LIN {X 0,Y 137.983,Z 516.99,A -85,B 0,C 180,E1 -24854.754,E2 -24854.754} C_VEL
LIN {X 0,Y 141.442,Z 522.73,A -85,B 0,C 180,E1 -24860.354,E2 -24860.354} C_VEL
LIN {X 0,Y 146.281,Z 527.08,A -85,B 0,C 180,E1 -24865.62,E2 -24865.62} C_VEL
LIN {X 0,Y 152.76,Z 530.196,A -85,B 0,C 180,E1 -24870.403,E2 -24870.403} C_VEL
LIN {X 0,Y 160.519,Z 532.095,A -85,B 0,C 180,E1 -24874.693,E2 -24874.693} C_VEL
LIN {X 0,Y 169.487,Z 532.782,A -85,B 0,C 180,E1 -24878.462,E2 -24878.462} C_VEL
LIN {X 0,Y 179.412,Z 532.227,A -85,B 0,C 180,E1 -24881.754,E2 -24881.754} C_VEL
LIN {X 0,Y 184.679,Z 531.482,A -85,B 0,C 180,E1 -24883.235,E2 -24883.235} C_VEL
LIN {X 0,Y 184.884,Z 531.53,A -85,B 0,C 180,E1 -24883.757,E2 -24883.757} C_VEL
LIN {X 0,Y 174.334,Z 533.909,A -85,B 0,C 180,E1 -24886.736,E2 -24886.736} C_VEL
LIN {X 0,Y 164.676,Z 535.155,A -85,B 0,C 180,E1 -24890.193,E2 -24890.193} C_VEL
LIN {X 0,Y 156.139,Z 535.296,A -85,B 0,C 180,E1 -24894.184,E2 -24894.184} C_VEL
LIN {X 0,Y 149.124,Z 534.399,A -85,B 0,C 180,E1 -24898.771,E2 -24898.771} C_VEL
LIN {X 0,Y 143.456,Z 532.415,A -85,B 0,C 180,E1 -24903.835,E2 -24903.835} C_VEL
LIN {X 0,Y 139.272,Z 529.177,A -85,B 0,C 180,E1 -24909.698,E2 -24909.698} C_VEL
LIN {X 0,Y 136.298,Z 533.394,A -85,B 0,C 180,E1 -24914.345,E2 -24914.345} C_VEL
LIN {X 0,Y 134.877,Z 535.787,A -85,B 0,C 180,E1 -24917.967,E2 -24917.967} C_VEL
LIN {X 0,Y 134.143,Z 537.216,A -85,B 0,C 180,E1 -24920.954,E2 -24920.954} C_VEL
LIN {X 0,Y 133.779,Z 538.232,A -85,B 0,C 180,E1 -24923.966,E2 -24923.966} C_VEL
LIN {X 0,Y 133.683,Z 538.88,A -85,B 0,C 180,E1 -24927.125,E2 -24927.125} C_VEL
LIN {X 0,Y 132.985,Z 539.095,A -85,B 0,C 180,E1 -24929.635,E2 -24929.635} C_VEL
LIN {X 0,Y 131.345,Z 538.952,A -85,B 0,C 180,E1 -24932.112,E2 -24932.112} C_VEL
LIN {X 0,Y 127.673,Z 537.738,A -85,B 0,C 180,E1 -24937.168,E2 -24937.168} C_VEL
LIN {X 0,Y 126.865,Z 536.758,A -85,B 0,C 180,E1 -24939.814,E2 -24939.814} C_VEL
LIN {X 0,Y 126.909,Z 536.327,A -85,B 0,C 180,E1 -24940.702,E2 -24940.702} C_VEL
LIN {X 0,Y 128.167,Z 533.463,A -85,B 0,C 180,E1 -24945.909,E2 -24945.909} C_VEL
LIN {X 0,Y 130.287,Z 529.76,A -85,B 0,C 180,E1 -24950.522,E2 -24950.522} C_VEL
LIN {X 0,Y 133.208,Z 524.928,A -85,B 0,C 180,E1 -24954.962,E2 -24954.962} C_VEL
LIN {X 0,Y 137.32,Z 517.944,A -85,B 0,C 180,E1 -24959.745,E2 -24959.745} C_VEL
LIN {X 0,Y 141.86,Z 509.751,A -85,B 0,C 180,E1 -24963.869,E2 -24963.869} C_VEL
LIN {X 0,Y 146.119,Z 501.674,A -85,B 0,C 180,E1 -24966.954,E2 -24966.954} C_VEL
LIN {X 0,Y 150.862,Z 491.823,A -85,B 0,C 180,E1 -24969.829,E2 -24969.829} C_VEL
LIN {X 0,Y 155.426,Z 480.689,A -85,B 0,C 180,E1 -24972.265,E2 -24972.265} C_VEL
LIN {X 0,Y 159.193,Z 469.804,A -85,B 0,C 180,E1 -24974.049,E2 -24974.049} C_VEL
LIN {X 0,Y 162.606,Z 457.774,A -85,B 0,C 180,E1 -24975.488,E2 -24975.488} C_VEL
LIN {X 0,Y 165.253,Z 444.892,A -85,B 0,C 180,E1 -24976.554,E2 -24976.554} C_VEL
LIN {X 0,Y 166.908,Z 431.8,A -85,B 0,C 180,E1 -24977.266,E2 -24977.266} C_VEL
LIN {X 0,Y 169.217,Z 398.153,A -85,B 0,C 180,E1 -24978.515,E2 -24978.515} C_VEL
LIN {X 0,Y 168.56,Z 385.284,A -85,B 0,C 180,E1 -24979.583,E2 -24979.583} C_VEL
LIN {X 0,Y 163.304,Z 375.445,A -85,B 0,C 180,E1 -24982.466,E2 -24982.466} C_VEL
LIN {X 0,Y 157.969,Z 366.553,A -85,B 0,C 180,E1 -24985.731,E2 -24985.731} C_VEL
LIN {X 0,Y 153.227,Z 359.41,A -85,B 0,C 180,E1 -24989.031,E2 -24989.031} C_VEL
LIN {X 0,Y 150.396,Z 355.476,A -85,B 0,C 180,E1 -24991.238,E2 -24991.238} C_VEL
LIN {X 0,Y 147.419,Z 351.407,A -85,B 0,C 180,E1 -24993.833,E2 -24993.833} C_VEL
LIN {X 0,Y 144.792,Z 348.208,A -85,B 0,C 180,E1 -24996.394,E2 -24996.394} C_VEL
LIN {X 0,Y 143.823,Z 346.644,A -85,B 0,C 180,E1 -24997.481,E2 -24997.481} C_VEL
LIN {X 0,Y 141.32,Z 344.263,A -85,B 0,C 180,E1 -25000.386,E2 -25000.386} C_VEL
LIN {X 0,Y 139.709,Z 341.234,A -85,B 0,C 180,E1 -25002.81,E2 -25002.81} C_VEL
LIN {X 0,Y 136.958,Z 339.298,A -85,B 0,C 180,E1 -25007.403,E2 -25007.403} C_VEL
LIN {X 0,Y 135.502,Z 336.05,A -85,B 0,C 180,E1 -25011.518,E2 -25011.518} C_VEL
LIN {X 0,Y 135.356,Z 335.408,A -85,B 0,C 180,E1 -25012.167,E2 -25012.167} C_VEL
LIN {X 0,Y 134.092,Z 334.839,A -85,B 0,C 180,E1 -25020,E2 -25020} C_VEL
LIN {X 0,Y 135.381,Z 335.546,A -85,B 0,C 180,E1 -25028.396,E2 -25028.396} C_VEL
LIN {X 0,Y 136.672,Z 338.936,A -85,B 0,C 180,E1 -25032.416,E2 -25032.416} C_VEL
LIN {X 0,Y 138.936,Z 340.918,A -85,B 0,C 180,E1 -25036.531,E2 -25036.531} C_VEL
LIN {X 0,Y 139.96,Z 341.514,A -85,B 0,C 180,E1 -25038.007,E2 -25038.007} C_VEL
LIN {X 0,Y 141.534,Z 344.542,A -85,B 0,C 180,E1 -25040.34,E2 -25040.34} C_VEL
LIN {X 0,Y 144.237,Z 347.153,A -85,B 0,C 180,E1 -25043.417,E2 -25043.417} C_VEL
LIN {X 0,Y 146.603,Z 350.647,A -85,B 0,C 180,E1 -25045.88,E2 -25045.88} C_VEL
LIN {X 0,Y 148.083,Z 352.258,A -85,B 0,C 180,E1 -25047.217,E2 -25047.217} C_VEL
LIN {X 0,Y 150.906,Z 356.018,A -85,B 0,C 180,E1 -25049.611,E2 -25049.611} C_VEL
LIN {X 0,Y 155.786,Z 363.227,A -85,B 0,C 180,E1 -25053.258,E2 -25053.258} C_VEL
LIN {X 0,Y 161.121,Z 371.713,A -85,B 0,C 180,E1 -25056.699,E2 -25056.699} C_VEL
LIN {X 0,Y 166.735,Z 381.737,A -85,B 0,C 180,E1 -25059.903,E2 -25059.903} C_VEL
LIN {X 0,Y 170.224,Z 388.868,A -85,B 0,C 180,E1 -25061.746,E2 -25061.746} C_VEL
LIN {X 0,Y 167.52,Z 425.77,A -85,B 0,C 180,E1 -25063.139,E2 -25063.139} C_VEL
LIN {X 0,Y 165.601,Z 439.061,A -85,B 0,C 180,E1 -25064.047,E2 -25064.047} C_VEL
LIN {X 0,Y 162.942,Z 451.365,A -85,B 0,C 180,E1 -25065.288,E2 -25065.288} C_VEL
LIN {X 0,Y 160.167,Z 461.584,A -85,B 0,C 180,E1 -25066.72,E2 -25066.72} C_VEL
LIN {X 0,Y 156.593,Z 471.955,A -85,B 0,C 180,E1 -25068.552,E2 -25068.552} C_VEL
LIN {X 0,Y 152.311,Z 482.567,A -85,B 0,C 180,E1 -25071.05,E2 -25071.05} C_VEL
LIN {X 0,Y 147.955,Z 492.24,A -85,B 0,C 180,E1 -25074.077,E2 -25074.077} C_VEL
LIN {X 0,Y 143.542,Z 500.604,A -85,B 0,C 180,E1 -25077.417,E2 -25077.417} C_VEL
LIN {X 0,Y 139.074,Z 508.063,A -85,B 0,C 180,E1 -25081.313,E2 -25081.313} C_VEL
LIN {X 0,Y 135.383,Z 514.04,A -85,B 0,C 180,E1 -25085.466,E2 -25085.466} C_VEL
LIN {X 0,Y 132.292,Z 518.76,A -85,B 0,C 180,E1 -25089.803,E2 -25089.803} C_VEL
LIN {X 0,Y 129.919,Z 522.361,A -85,B 0,C 180,E1 -25094.311,E2 -25094.311} C_VEL
LIN {X 0,Y 128.741,Z 524.212,A -85,B 0,C 180,E1 -25097.391,E2 -25097.391} C_VEL
LIN {X 0,Y 127.826,Z 525.621,A -85,B 0,C 180,E1 -25100.509,E2 -25100.509} C_VEL
LIN {X 0,Y 126.857,Z 527.214,A -85,B 0,C 180,E1 -25106.827,E2 -25106.827} C_VEL
LIN {X 0,Y 126.763,Z 527.441,A -85,B 0,C 180,E1 -25110.003,E2 -25110.003} C_VEL
LIN {X 0,Y 127.085,Z 526.871,A -85,B 0,C 180,E1 -25115.478,E2 -25115.478} C_VEL
LIN {X 0,Y 127.815,Z 525.69,A -85,B 0,C 180,E1 -25119.498,E2 -25119.498} C_VEL
LIN {X 0,Y 128.715,Z 524.32,A -85,B 0,C 180,E1 -25122.619,E2 -25122.619} C_VEL
LIN {X 0,Y 130.56,Z 521.447,A -85,B 0,C 180,E1 -25127.224,E2 -25127.224} C_VEL
LIN {X 0,Y 133.185,Z 517.529,A -85,B 0,C 180,E1 -25131.681,E2 -25131.681} C_VEL
LIN {X 0,Y 136.479,Z 512.452,A -85,B 0,C 180,E1 -25135.961,E2 -25135.961} C_VEL
LIN {X 0,Y 140.425,Z 506.047,A -85,B 0,C 180,E1 -25140.035,E2 -25140.035} C_VEL
LIN {X 0,Y 145.115,Z 498.061,A -85,B 0,C 180,E1 -25143.848,E2 -25143.848} C_VEL
LIN {X 0,Y 149.172,Z 489.824,A -85,B 0,C 180,E1 -25146.958,E2 -25146.958} C_VEL
LIN {X 0,Y 153.639,Z 479.82,A -85,B 0,C 180,E1 -25149.825,E2 -25149.825} C_VEL
LIN {X 0,Y 157.58,Z 469.857,A -85,B 0,C 180,E1 -25151.993,E2 -25151.993} C_VEL
LIN {X 0,Y 161.097,Z 458.996,A -85,B 0,C 180,E1 -25153.836,E2 -25153.836} C_VEL
LIN {X 0,Y 164.233,Z 446.902,A -85,B 0,C 180,E1 -25155.354,E2 -25155.354} C_VEL
LIN {X 0,Y 166.651,Z 433.829,A -85,B 0,C 180,E1 -25156.511,E2 -25156.511} C_VEL
LIN {X 0,Y 168.152,Z 421.523,A -85,B 0,C 180,E1 -25157.195,E2 -25157.195} C_VEL
LIN {X 0,Y 170.406,Z 389.046,A -85,B 0,C 180,E1 -25158.395,E2 -25158.395} C_VEL
LIN {X 0,Y 165.265,Z 378.802,A -85,B 0,C 180,E1 -25161.152,E2 -25161.152} C_VEL
LIN {X 0,Y 160.009,Z 369.693,A -85,B 0,C 180,E1 -25164.252,E2 -25164.252} C_VEL
LIN {X 0,Y 155.37,Z 362.549,A -85,B 0,C 180,E1 -25167.317,E2 -25167.317} C_VEL
LIN {X 0,Y 153.571,Z 359.786,A -85,B 0,C 180,E1 -25168.63,E2 -25168.63} C_VEL
LIN {X 0,Y 153.009,Z 359.751,A -85,B 0,C 180,E1 -25168.982,E2 -25168.982} C_VEL
LIN {X 0,Y 151.499,Z 361.411,A -85,B 0,C 180,E1 -25169.798,E2 -25169.798} C_VEL
LIN {X 0,Y 147.778,Z 373.075,A -85,B 0,C 180,E1 -25171.215,E2 -25171.215} C_VEL
LIN {X 0,Y 145.671,Z 378.207,A -85,B 0,C 180,E1 -25172.233,E2 -25172.233} C_VEL
LIN {X 0,Y 143.605,Z 381.544,A -85,B 0,C 180,E1 -25173.484,E2 -25173.484} C_VEL
LIN {X 0,Y 142.496,Z 382.609,A -85,B 0,C 180,E1 -25174.277,E2 -25174.277} C_VEL
LIN {X 0,Y 138.592,Z 397.916,A -85,B 0,C 180,E1 -25175.899,E2 -25175.899} C_VEL
LIN {X 0,Y 135.86,Z 407.043,A -85,B 0,C 180,E1 -25177.372,E2 -25177.372} C_VEL
LIN {X 0,Y 134.347,Z 410.966,A -85,B 0,C 180,E1 -25178.419,E2 -25178.419} C_VEL
LIN {X 0,Y 133.86,Z 411.757,A -85,B 0,C 180,E1 -25178.841,E2 -25178.841} C_VEL
LIN {X 0,Y 133.459,Z 411.859,A -85,B 0,C 180,E1 -25179.279,E2 -25179.279} C_VEL
LIN {X 0,Y 133.201,Z 410.793,A -85,B 0,C 180,E1 -25179.741,E2 -25179.741} C_VEL
LIN {X 0,Y 133.317,Z 407.838,A -85,B 0,C 180,E1 -25180.162,E2 -25180.162} C_VEL
LIN {X 0,Y 132.531,Z 426.85,A -85,B 0,C 180,E1 -25182.345,E2 -25182.345} C_VEL
LIN {X 0,Y 131.767,Z 440.893,A -85,B 0,C 180,E1 -25184.533,E2 -25184.533} C_VEL
LIN {X 0,Y 131.039,Z 452.449,A -85,B 0,C 180,E1 -25186.876,E2 -25186.876} C_VEL
LIN {X 0,Y 130.192,Z 465.708,A -85,B 0,C 180,E1 -25190.288,E2 -25190.288} C_VEL
LIN {X 0,Y 129.673,Z 476.575,A -85,B 0,C 180,E1 -25193.777,E2 -25193.777} C_VEL
LIN {X 0,Y 129.296,Z 486.462,A -85,B 0,C 180,E1 -25197.663,E2 -25197.663} C_VEL
LIN {X 0,Y 129.201,Z 494.658,A -85,B 0,C 180,E1 -25201.558,E2 -25201.558} C_VEL
LIN {X 0,Y 129.288,Z 502.752,A -85,B 0,C 180,E1 -25206.241,E2 -25206.241} C_VEL
LIN {X 0,Y 130.06,Z 510.449,A -85,B 0,C 180,E1 -25211.691,E2 -25211.691} C_VEL
LIN {X 0,Y 132.13,Z 516.795,A -85,B 0,C 180,E1 -25217.009,E2 -25217.009} C_VEL
LIN {X 0,Y 136.037,Z 522.64,A -85,B 0,C 180,E1 -25222.797,E2 -25222.797} C_VEL
LIN {X 0,Y 139.975,Z 526.09,A -85,B 0,C 180,E1 -25226.864,E2 -25226.864} C_VEL
LIN {X 0,Y 146.71,Z 529.673,A -85,B 0,C 180,E1 -25231.799,E2 -25231.799} C_VEL
LIN {X 0,Y 154.737,Z 532.05,A -85,B 0,C 180,E1 -25236.189,E2 -25236.189} C_VEL
LIN {X 0,Y 163.997,Z 533.24,A -85,B 0,C 180,E1 -25240.002,E2 -25240.002} C_VEL
LIN {X 0,Y 174.202,Z 533.221,A -85,B 0,C 180,E1 -25243.302,E2 -25243.302} C_VEL
LIN {X 0,Y 174.544,Z 533.221,A -85,B 0,C 180,E1 -25243.547,E2 -25243.547} C_VEL
LIN {X 0,Y 164.125,Z 534.493,A -85,B 0,C 180,E1 -25246.751,E2 -25246.751} C_VEL
LIN {X 0,Y 153.064,Z 534.613,A -85,B 0,C 180,E1 -25251.312,E2 -25251.312} C_VEL
LIN {X 0,Y 146.693,Z 533.865,A -85,B 0,C 180,E1 -25254.903,E2 -25254.903} C_VEL
LIN {X 0,Y 140.065,Z 532.02,A -85,B 0,C 180,E1 -25259.88,E2 -25259.88} C_VEL
LIN {X 0,Y 134.974,Z 529.091,A -85,B 0,C 180,E1 -25265.38,E2 -25265.38} C_VEL
LIN {X 0,Y 133.476,Z 527.79,A -85,B 0,C 180,E1 -25267.657,E2 -25267.657} C_VEL
LIN {X 0,Y 129.895,Z 532.5,A -85,B 0,C 180,E1 -25272.685,E2 -25272.685} C_VEL
LIN {X 0,Y 127.936,Z 535.47,A -85,B 0,C 180,E1 -25277.303,E2 -25277.303} C_VEL
LIN {X 0,Y 127.137,Z 536.899,A -85,B 0,C 180,E1 -25280.451,E2 -25280.451} C_VEL
LIN {X 0,Y 126.721,Z 537.916,A -85,B 0,C 180,E1 -25283.628,E2 -25283.628} C_VEL
LIN {X 0,Y 126.611,Z 538.647,A -85,B 0,C 180,E1 -25287.651,E2 -25287.651} C_VEL
LIN {X 0,Y 126.759,Z 538.767,A -85,B 0,C 180,E1 -25289.997,E2 -25289.997} C_VEL
LIN {X 0,Y 126.546,Z 538.522,A -85,B 0,C 180,E1 -25293.18,E2 -25293.18} C_VEL
LIN {X 0,Y 126.756,Z 536.845,A -85,B 0,C 180,E1 -25299.571,E2 -25299.571} C_VEL
LIN {X 0,Y 126.909,Z 536.327,A -85,B 0,C 180,E1 -25300.702,E2 -25300.702} C_VEL
LIN {X 0,Y 126.775,Z 535.087,A -85,B 0,C 180,E1 -25303.305,E2 -25303.305} C_VEL
LIN {X 0,Y 125.297,Z 532.462,A -85,B 0,C 180,E1 -25307.605,E2 -25307.605} C_VEL
LIN {X 0,Y 124.449,Z 529.896,A -85,B 0,C 180,E1 -25311.042,E2 -25311.042} C_VEL
LIN {X 0,Y 124.853,Z 527.661,A -85,B 0,C 180,E1 -25313.555,E2 -25313.555} C_VEL
LIN {X 0,Y 125.292,Z 526.84,A -85,B 0,C 180,E1 -25314.356,E2 -25314.356} C_VEL
LIN {X 0,Y 129.229,Z 520.714,A -85,B 0,C 180,E1 -25319.301,E2 -25319.301} C_VEL
LIN {X 0,Y 133.556,Z 513.613,A -85,B 0,C 180,E1 -25323.537,E2 -25323.537} C_VEL
LIN {X 0,Y 138.648,Z 504.783,A -85,B 0,C 180,E1 -25327.461,E2 -25327.461} C_VEL
LIN {X 0,Y 143.436,Z 495.72,A -85,B 0,C 180,E1 -25330.479,E2 -25330.479} C_VEL
LIN {X 0,Y 148.106,Z 485.642,A -85,B 0,C 180,E1 -25333.006,E2 -25333.006} C_VEL
LIN {X 0,Y 152.465,Z 474.478,A -85,B 0,C 180,E1 -25335.127,E2 -25335.127} C_VEL
LIN {X 0,Y 156.222,Z 462.931,A -85,B 0,C 180,E1 -25336.734,E2 -25336.734} C_VEL
LIN {X 0,Y 159.321,Z 450.322,A -85,B 0,C 180,E1 -25337.985,E2 -25337.985} C_VEL
LIN {X 0,Y 161.652,Z 436.707,A -85,B 0,C 180,E1 -25338.862,E2 -25338.862} C_VEL
LIN {X 0,Y 164.022,Z 407.003,A -85,B 0,C 180,E1 -25340.003,E2 -25340.003} C_VEL
LIN {X 0,Y 164.518,Z 398.539,A -85,B 0,C 180,E1 -25340.36,E2 -25340.36} C_VEL
LIN {X 0,Y 163.994,Z 388.51,A -85,B 0,C 180,E1 -25341.257,E2 -25341.257} C_VEL
LIN {X 0,Y 158.892,Z 378.792,A -85,B 0,C 180,E1 -25344.317,E2 -25344.317} C_VEL
LIN {X 0,Y 153.534,Z 369.735,A -85,B 0,C 180,E1 -25347.947,E2 -25347.947} C_VEL
LIN {X 0,Y 149.787,Z 364.14,A -85,B 0,C 180,E1 -25350.822,E2 -25350.822} C_VEL
LIN {X 0,Y 147.92,Z 361.462,A -85,B 0,C 180,E1 -25352.403,E2 -25352.403} C_VEL
LIN {X 0,Y 145.368,Z 357.807,A -85,B 0,C 180,E1 -25354.783,E2 -25354.783} C_VEL
LIN {X 0,Y 142.706,Z 354.313,A -85,B 0,C 180,E1 -25357.575,E2 -25357.575} C_VEL
LIN {X 0,Y 141.994,Z 353.199,A -85,B 0,C 180,E1 -25358.422,E2 -25358.422} C_VEL
LIN {X 0,Y 139.451,Z 350.415,A -85,B 0,C 180,E1 -25361.64,E2 -25361.64} C_VEL
LIN {X 0,Y 138.378,Z 348.166,A -85,B 0,C 180,E1 -25363.4,E2 -25363.4} C_VEL
LIN {X 0,Y 135.587,Z 345.861,A -85,B 0,C 180,E1 -25368.457,E2 -25368.457} C_VEL
LIN {X 0,Y 134.268,Z 342.408,A -85,B 0,C 180,E1 -25372.859,E2 -25372.859} C_VEL
LIN {X 0,Y 133.228,Z 341.881,A -85,B 0,C 180,E1 -25380,E2 -25380} C_VEL
LIN {X 0,Y 134.331,Z 342.692,A -85,B 0,C 180,E1 -25387.894,E2 -25387.894} C_VEL
LIN {X 0,Y 135.726,Z 346.121,A -85,B 0,C 180,E1 -25392.333,E2 -25392.333} C_VEL
LIN {X 0,Y 138.44,Z 348.337,A -85,B 0,C 180,E1 -25397.162,E2 -25397.162} C_VEL
LIN {X 0,Y 140.391,Z 351.729,A -85,B 0,C 180,E1 -25400.114,E2 -25400.114} C_VEL
LIN {X 0,Y 142.392,Z 353.705,A -85,B 0,C 180,E1 -25402.49,E2 -25402.49} C_VEL
LIN {X 0,Y 144.806,Z 357.248,A -85,B 0,C 180,E1 -25405.13,E2 -25405.13} C_VEL
LIN {X 0,Y 146.115,Z 358.845,A -85,B 0,C 180,E1 -25406.389,E2 -25406.389} C_VEL
LIN {X 0,Y 149.396,Z 363.613,A -85,B 0,C 180,E1 -25409.311,E2 -25409.311} C_VEL
LIN {X 0,Y 152.868,Z 368.804,A -85,B 0,C 180,E1 -25412.027,E2 -25412.027} C_VEL
LIN {X 0,Y 157.952,Z 377.189,A -85,B 0,C 180,E1 -25415.539,E2 -25415.539} C_VEL
LIN {X 0,Y 163.364,Z 387.261,A -85,B 0,C 180,E1 -25418.839,E2 -25418.839} C_VEL
LIN {X 0,Y 165.441,Z 391.583,A -85,B 0,C 180,E1 -25420.019,E2 -25420.019} C_VEL
LIN {X 0,Y 162.744,Z 426.104,A -85,B 0,C 180,E1 -25421.319,E2 -25421.319} C_VEL
LIN {X 0,Y 160.761,Z 439.35,A -85,B 0,C 180,E1 -25422.234,E2 -25422.234} C_VEL
LIN {X 0,Y 157.996,Z 451.663,A -85,B 0,C 180,E1 -25423.484,E2 -25423.484} C_VEL
LIN {X 0,Y 155.097,Z 461.888,A -85,B 0,C 180,E1 -25424.93,E2 -25424.93} C_VEL
LIN {X 0,Y 151.362,Z 472.264,A -85,B 0,C 180,E1 -25426.779,E2 -25426.779} C_VEL
LIN {X 0,Y 146.851,Z 482.88,A -85,B 0,C 180,E1 -25429.307,E2 -25429.307} C_VEL
LIN {X 0,Y 142.841,Z 491.293,A -85,B 0,C 180,E1 -25431.927,E2 -25431.927} C_VEL
LIN {X 0,Y 138.465,Z 499.472,A -85,B 0,C 180,E1 -25435.183,E2 -25435.183} C_VEL
LIN {X 0,Y 133.638,Z 507.264,A -85,B 0,C 180,E1 -25439.157,E2 -25439.157} C_VEL
LIN {X 0,Y 130.198,Z 512.522,A -85,B 0,C 180,E1 -25442.692,E2 -25442.692} C_VEL
LIN {X 0,Y 126.678,Z 517.653,A -85,B 0,C 180,E1 -25447.152,E2 -25447.152} C_VEL
LIN {X 0,Y 123.861,Z 521.615,A -85,B 0,C 180,E1 -25451.819,E2 -25451.819} C_VEL
LIN {X 0,Y 121.837,Z 524.529,A -85,B 0,C 180,E1 -25456.663,E2 -25456.663} C_VEL
LIN {X 0,Y 120.845,Z 525.937,A -85,B 0,C 180,E1 -25459.956,E2 -25459.956} C_VEL
LIN {X 0,Y 119.791,Z 527.531,A -85,B 0,C 180,E1 -25466.64,E2 -25466.64} C_VEL
LIN {X 0,Y 119.67,Z 527.758,A -85,B 0,C 180,E1 -25470.003,E2 -25470.003} C_VEL
LIN {X 0,Y 119.911,Z 527.35,A -85,B 0,C 180,E1 -25474.878,E2 -25474.878} C_VEL
LIN {X 0,Y 120.815,Z 526.006,A -85,B 0,C 180,E1 -25480.054,E2 -25480.054} C_VEL
LIN {X 0,Y 121.797,Z 524.637,A -85,B 0,C 180,E1 -25483.348,E2 -25483.348} C_VEL
LIN {X 0,Y 123.807,Z 521.762,A -85,B 0,C 180,E1 -25488.196,E2 -25488.196} C_VEL
LIN {X 0,Y 126.606,Z 517.844,A -85,B 0,C 180,E1 -25492.869,E2 -25492.869} C_VEL
LIN {X 0,Y 130.139,Z 512.765,A -85,B 0,C 180,E1 -25497.328,E2 -25497.328} C_VEL
LIN {X 0,Y 134.337,Z 506.359,A -85,B 0,C 180,E1 -25501.548,E2 -25501.548} C_VEL
LIN {X 0,Y 139.286,Z 498.371,A -85,B 0,C 180,E1 -25505.472,E2 -25505.472} C_VEL
LIN {X 0,Y 143.943,Z 489.359,A -85,B 0,C 180,E1 -25508.918,E2 -25508.918} C_VEL
LIN {X 0,Y 148.773,Z 478.982,A -85,B 0,C 180,E1 -25511.859,E2 -25511.859} C_VEL
LIN {X 0,Y 152.929,Z 468.772,A -85,B 0,C 180,E1 -25514.037,E2 -25514.037} C_VEL
LIN {X 0,Y 156.613,Z 457.517,A -85,B 0,C 180,E1 -25515.893,E2 -25515.893} C_VEL
LIN {X 0,Y 159.628,Z 445.943,A -85,B 0,C 180,E1 -25517.286,E2 -25517.286} C_VEL
LIN {X 0,Y 161.978,Z 433.307,A -85,B 0,C 180,E1 -25518.39,E2 -25518.39} C_VEL
LIN {X 0,Y 163.577,Z 419.844,A -85,B 0,C 180,E1 -25519.098,E2 -25519.098} C_VEL
LIN {X 0,Y 165.6,Z 391.684,A -85,B 0,C 180,E1 -25520.141,E2 -25520.141} C_VEL
LIN {X 0,Y 160.783,Z 382.051,A -85,B 0,C 180,E1 -25522.956,E2 -25522.956} C_VEL
LIN {X 0,Y 155.848,Z 373.35,A -85,B 0,C 180,E1 -25526.152,E2 -25526.152} C_VEL
LIN {X 0,Y 153.058,Z 369.064,A -85,B 0,C 180,E1 -25528.126,E2 -25528.126} C_VEL
LIN {X 0,Y 149.53,Z 378.939,A -85,B 0,C 180,E1 -25529.456,E2 -25529.456} C_VEL
LIN {X 0,Y 147.014,Z 384.13,A -85,B 0,C 180,E1 -25530.659,E2 -25530.659} C_VEL
LIN {X 0,Y 144.614,Z 387.577,A -85,B 0,C 180,E1 -25532.049,E2 -25532.049} C_VEL
LIN {X 0,Y 140.205,Z 403.592,A -85,B 0,C 180,E1 -25533.795,E2 -25533.795} C_VEL
LIN {X 0,Y 137.254,Z 412.423,A -85,B 0,C 180,E1 -25535.329,E2 -25535.329} C_VEL
LIN {X 0,Y 135.386,Z 416.509,A -85,B 0,C 180,E1 -25536.581,E2 -25536.581} C_VEL
LIN {X 0,Y 133.899,Z 418.455,A -85,B 0,C 180,E1 -25537.836,E2 -25537.836} C_VEL
LIN {X 0,Y 133.547,Z 418.68,A -85,B 0,C 180,E1 -25538.181,E2 -25538.181} C_VEL
LIN {X 0,Y 130.543,Z 429.71,A -85,B 0,C 180,E1 -25539.619,E2 -25539.619} C_VEL
LIN {X 0,Y 128.161,Z 435.709,A -85,B 0,C 180,E1 -25540.906,E2 -25540.906} C_VEL
LIN {X 0,Y 126.348,Z 439.161,A -85,B 0,C 180,E1 -25542.14,E2 -25542.14} C_VEL
LIN {X 0,Y 125.101,Z 440.725,A -85,B 0,C 180,E1 -25543.382,E2 -25543.382} C_VEL
LIN {X 0,Y 124.702,Z 440.196,A -85,B 0,C 180,E1 -25544.287,E2 -25544.287} C_VEL
LIN {X 0,Y 124.922,Z 438.313,A -85,B 0,C 180,E1 -25544.764,E2 -25544.764} C_VEL
LIN {X 0,Y 124.122,Z 452.23,A -85,B 0,C 180,E1 -25547.741,E2 -25547.741} C_VEL
LIN {X 0,Y 123.392,Z 465.645,A -85,B 0,C 180,E1 -25551.401,E2 -25551.401} C_VEL
LIN {X 0,Y 122.918,Z 476.449,A -85,B 0,C 180,E1 -25555.08,E2 -25555.08} C_VEL
LIN {X 0,Y 122.616,Z 486.247,A -85,B 0,C 180,E1 -25559.179,E2 -25559.179} C_VEL
LIN {X 0,Y 122.6,Z 494.382,A -85,B 0,C 180,E1 -25563.286,E2 -25563.286} C_VEL
LIN {X 0,Y 122.86,Z 502.425,A -85,B 0,C 180,E1 -25568.222,E2 -25568.222} C_VEL
LIN {X 0,Y 123.989,Z 510.25,A -85,B 0,C 180,E1 -25574.068,E2 -25574.068} C_VEL
LIN {X 0,Y 126.481,Z 516.495,A -85,B 0,C 180,E1 -25579.475,E2 -25579.475} C_VEL
LIN {X 0,Y 130.973,Z 522.427,A -85,B 0,C 180,E1 -25585.422,E2 -25585.422} C_VEL
LIN {X 0,Y 137.097,Z 527.06,A -85,B 0,C 180,E1 -25590.839,E2 -25590.839} C_VEL
LIN {X 0,Y 144.76,Z 530.49,A -85,B 0,C 180,E1 -25595.633,E2 -25595.633} C_VEL
LIN {X 0,Y 153.725,Z 532.757,A -85,B 0,C 180,E1 -25599.796,E2 -25599.796} C_VEL
LIN {X 0,Y 163.761,Z 533.864,A -85,B 0,C 180,E1 -25603.366,E2 -25603.366} C_VEL
LIN {X 0,Y 154.093,Z 534.071,A -85,B 0,C 180,E1 -25606.829,E2 -25606.829} C_VEL
LIN {X 0,Y 144.99,Z 533.277,A -85,B 0,C 180,E1 -25610.936,E2 -25610.936} C_VEL
LIN {X 0,Y 137.406,Z 531.542,A -85,B 0,C 180,E1 -25615.759,E2 -25615.759} C_VEL
LIN {X 0,Y 131.294,Z 528.778,A -85,B 0,C 180,E1 -25621.196,E2 -25621.196} C_VEL
LIN {X 0,Y 127.967,Z 526.275,A -85,B 0,C 180,E1 -25625.348,E2 -25625.348} C_VEL
LIN {X 0,Y 124.089,Z 530.949,A -85,B 0,C 180,E1 -25630.131,E2 -25630.131} C_VEL
LIN {X 0,Y 122.322,Z 533.263,A -85,B 0,C 180,E1 -25633.302,E2 -25633.302} C_VEL
LIN {X 0,Y 121.024,Z 535.154,A -85,B 0,C 180,E1 -25636.565,E2 -25636.565} C_VEL
LIN {X 0,Y 120.132,Z 536.582,A -85,B 0,C 180,E1 -25639.889,E2 -25639.889} C_VEL
LIN {X 0,Y 119.665,Z 537.599,A -85,B 0,C 180,E1 -25643.251,E2 -25643.251} C_VEL
LIN {X 0,Y 119.539,Z 538.363,A -85,B 0,C 180,E1 -25648.14,E2 -25648.14} C_VEL
LIN {X 0,Y 119.528,Z 538.366,A -85,B 0,C 180,E1 -25651.68,E2 -25651.68} C_VEL
LIN {X 0,Y 119.414,Z 537.56,A -85,B 0,C 180,E1 -25656.756,E2 -25656.756} C_VEL
LIN {X 0,Y 119.83,Z 536.184,A -85,B 0,C 180,E1 -25660.927,E2 -25660.927} C_VEL
LIN {X 0,Y 121.304,Z 533.143,A -85,B 0,C 180,E1 -25666.836,E2 -25666.836} C_VEL
LIN {X 0,Y 123.626,Z 529.441,A -85,B 0,C 180,E1 -25671.682,E2 -25671.682} C_VEL
LIN {X 0,Y 125.292,Z 526.84,A -85,B 0,C 180,E1 -25674.356,E2 -25674.356} C_VEL
LIN {X 0,Y 126.313,Z 524.282,A -85,B 0,C 180,E1 -25676.74,E2 -25676.74} C_VEL
LIN {X 0,Y 126.65,Z 519.66,A -85,B 0,C 180,E1 -25680.72,E2 -25680.72} C_VEL
LIN {X 0,Y 127.452,Z 514.492,A -85,B 0,C 180,E1 -25684.512,E2 -25684.512} C_VEL
LIN {X 0,Y 129.13,Z 510.958,A -85,B 0,C 180,E1 -25686.508,E2 -25686.508} C_VEL
LIN {X 0,Y 134.023,Z 502.811,A -85,B 0,C 180,E1 -25689.965,E2 -25689.965} C_VEL
LIN {X 0,Y 139.682,Z 492.255,A -85,B 0,C 180,E1 -25693.273,E2 -25693.273} C_VEL
LIN {X 0,Y 144.652,Z 481.473,A -85,B 0,C 180,E1 -25695.773,E2 -25695.773} C_VEL
LIN {X 0,Y 149.329,Z 469.194,A -85,B 0,C 180,E1 -25697.834,E2 -25697.834} C_VEL
LIN {X 0,Y 152.982,Z 457.178,A -85,B 0,C 180,E1 -25699.285,E2 -25699.285} C_VEL
LIN {X 0,Y 155.84,Z 444.394,A -85,B 0,C 180,E1 -25700.333,E2 -25700.333} C_VEL
LIN {X 0,Y 157.667,Z 430.813,A -85,B 0,C 180,E1 -25701.081,E2 -25701.081} C_VEL
LIN {X 0,Y 160.012,Z 399.892,A -85,B 0,C 180,E1 -25702.236,E2 -25702.236} C_VEL
LIN {X 0,Y 159.694,Z 392.035,A -85,B 0,C 180,E1 -25702.949,E2 -25702.949} C_VEL
LIN {X 0,Y 154.992,Z 382.858,A -85,B 0,C 180,E1 -25706.03,E2 -25706.03} C_VEL
LIN {X 0,Y 150.219,Z 374.668,A -85,B 0,C 180,E1 -25709.552,E2 -25709.552} C_VEL
LIN {X 0,Y 146.257,Z 368.327,A -85,B 0,C 180,E1 -25712.935,E2 -25712.935} C_VEL
LIN {X 0,Y 143.037,Z 363.842,A -85,B 0,C 180,E1 -25716.087,E2 -25716.087} C_VEL
LIN {X 0,Y 140.149,Z 359.718,A -85,B 0,C 180,E1 -25719.45,E2 -25719.45} C_VEL
LIN {X 0,Y 137.596,Z 356.471,A -85,B 0,C 180,E1 -25723.016,E2 -25723.016} C_VEL
LIN {X 0,Y 136.731,Z 354.84,A -85,B 0,C 180,E1 -25724.536,E2 -25724.536} C_VEL
LIN {X 0,Y 134.318,Z 352.511,A -85,B 0,C 180,E1 -25729.384,E2 -25729.384} C_VEL
LIN {X 0,Y 133.202,Z 349.397,A -85,B 0,C 180,E1 -25733.563,E2 -25733.563} C_VEL
LIN {X 0,Y 132.363,Z 348.925,A -85,B 0,C 180,E1 -25740,E2 -25740} C_VEL
LIN {X 0,Y 133.273,Z 349.6,A -85,B 0,C 180,E1 -25747.222,E2 -25747.222} C_VEL
LIN {X 0,Y 134.547,Z 352.949,A -85,B 0,C 180,E1 -25751.678,E2 -25751.678} C_VEL
LIN {X 0,Y 137.011,Z 355.175,A -85,B 0,C 180,E1 -25756.387,E2 -25756.387} C_VEL
LIN {X 0,Y 138.908,Z 358.473,A -85,B 0,C 180,E1 -25759.415,E2 -25759.415} C_VEL
LIN {X 0,Y 140.731,Z 360.465,A -85,B 0,C 180,E1 -25761.719,E2 -25761.719} C_VEL
LIN {X 0,Y 143.307,Z 364.12,A -85,B 0,C 180,E1 -25764.636,E2 -25764.636} C_VEL
LIN {X 0,Y 146.88,Z 369.431,A -85,B 0,C 180,E1 -25768.096,E2 -25768.096} C_VEL
LIN {X 0,Y 150.191,Z 374.647,A -85,B 0,C 180,E1 -25770.882,E2 -25770.882} C_VEL
LIN {X 0,Y 154.992,Z 382.911,A -85,B 0,C 180,E1 -25774.429,E2 -25774.429} C_VEL
LIN {X 0,Y 159.72,Z 392.059,A -85,B 0,C 180,E1 -25777.521,E2 -25777.521} C_VEL
LIN {X 0,Y 160.741,Z 394.25,A -85,B 0,C 180,E1 -25778.153,E2 -25778.153} C_VEL
LIN {X 0,Y 158.103,Z 426.795,A -85,B 0,C 180,E1 -25779.411,E2 -25779.411} C_VEL
LIN {X 0,Y 156.087,Z 439.639,A -85,B 0,C 180,E1 -25780.308,E2 -25780.308} C_VEL
LIN {X 0,Y 153.201,Z 451.963,A -85,B 0,C 180,E1 -25781.559,E2 -25781.559} C_VEL
LIN {X 0,Y 150.186,Z 462.193,A -85,B 0,C 180,E1 -25783.019,E2 -25783.019} C_VEL
LIN {X 0,Y 146.289,Z 472.572,A -85,B 0,C 180,E1 -25784.882,E2 -25784.882} C_VEL
LIN {X 0,Y 141.551,Z 483.192,A -85,B 0,C 180,E1 -25787.435,E2 -25787.435} C_VEL
LIN {X 0,Y 137.099,Z 492.034,A -85,B 0,C 180,E1 -25790.258,E2 -25790.258} C_VEL
LIN {X 0,Y 131.821,Z 501.234,A -85,B 0,C 180,E1 -25794.098,E2 -25794.098} C_VEL
LIN {X 0,Y 126.808,Z 508.695,A -85,B 0,C 180,E1 -25798.234,E2 -25798.234} C_VEL
LIN {X 0,Y 122.605,Z 514.674,A -85,B 0,C 180,E1 -25802.708,E2 -25802.708} C_VEL
LIN {X 0,Y 119.055,Z 519.395,A -85,B 0,C 180,E1 -25807.44,E2 -25807.44} C_VEL
LIN {X 0,Y 116.32,Z 522.995,A -85,B 0,C 180,E1 -25812.42,E2 -25812.42} C_VEL
LIN {X 0,Y 114.933,Z 524.846,A -85,B 0,C 180,E1 -25815.846,E2 -25815.846} C_VEL
LIN {X 0,Y 113.865,Z 526.255,A -85,B 0,C 180,E1 -25819.333,E2 -25819.333} C_VEL
LIN {X 0,Y 112.707,Z 527.848,A -85,B 0,C 180,E1 -25826.429,E2 -25826.429} C_VEL
LIN {X 0,Y 112.578,Z 528.075,A -85,B 0,C 180,E1 -25830.004,E2 -25830.004} C_VEL
LIN {X 0,Y 112.778,Z 527.771,A -85,B 0,C 180,E1 -25834.381,E2 -25834.381} C_VEL
LIN {X 0,Y 113.844,Z 526.322,A -85,B 0,C 180,E1 -25840.676,E2 -25840.676} C_VEL
LIN {X 0,Y 114.892,Z 524.953,A -85,B 0,C 180,E1 -25844.167,E2 -25844.167} C_VEL
LIN {X 0,Y 117.101,Z 522.076,A -85,B 0,C 180,E1 -25849.278,E2 -25849.278} C_VEL
LIN {X 0,Y 120.095,Z 518.159,A -85,B 0,C 180,E1 -25854.186,E2 -25854.186} C_VEL
LIN {X 0,Y 123.861,Z 513.079,A -85,B 0,C 180,E1 -25858.839,E2 -25858.839} C_VEL
LIN {X 0,Y 128.353,Z 506.67,A -85,B 0,C 180,E1 -25863.203,E2 -25863.203} C_VEL
LIN {X 0,Y 133.572,Z 498.681,A -85,B 0,C 180,E1 -25867.238,E2 -25867.238} C_VEL
LIN {X 0,Y 138.427,Z 489.793,A -85,B 0,C 180,E1 -25870.722,E2 -25870.722} C_VEL
LIN {X 0,Y 143.041,Z 480.428,A -85,B 0,C 180,E1 -25873.464,E2 -25873.464} C_VEL
LIN {X 0,Y 147.908,Z 469.072,A -85,B 0,C 180,E1 -25875.949,E2 -25875.949} C_VEL
LIN {X 0,Y 151.761,Z 457.808,A -85,B 0,C 180,E1 -25877.816,E2 -25877.816} C_VEL
LIN {X 0,Y 155.186,Z 444.985,A -85,B 0,C 180,E1 -25879.342,E2 -25879.342} C_VEL
LIN {X 0,Y 157.623,Z 431.918,A -85,B 0,C 180,E1 -25880.435,E2 -25880.435} C_VEL
LIN {X 0,Y 159.241,Z 417.59,A -85,B 0,C 180,E1 -25881.113,E2 -25881.113} C_VEL
LIN {X 0,Y 160.986,Z 395.107,A -85,B 0,C 180,E1 -25881.919,E2 -25881.919} C_VEL
LIN {X 0,Y 160.576,Z 393.662,A -85,B 0,C 180,E1 -25882.211,E2 -25882.211} C_VEL
LIN {X 0,Y 156.389,Z 385.283,A -85,B 0,C 180,E1 -25884.905,E2 -25884.905} C_VEL
LIN {X 0,Y 153.558,Z 380.099,A -85,B 0,C 180,E1 -25886.883,E2 -25886.883} C_VEL
LIN {X 0,Y 153.323,Z 380.07,A -85,B 0,C 180,E1 -25887.021,E2 -25887.021} C_VEL
LIN {X 0,Y 150.567,Z 386.301,A -85,B 0,C 180,E1 -25888.127,E2 -25888.127} C_VEL
LIN {X 0,Y 147.637,Z 391.183,A -85,B 0,C 180,E1 -25889.554,E2 -25889.554} C_VEL
LIN {X 0,Y 146.9,Z 392.446,A -85,B 0,C 180,E1 -25889.929,E2 -25889.929} C_VEL
LIN {X 0,Y 142.602,Z 407.227,A -85,B 0,C 180,E1 -25891.507,E2 -25891.507} C_VEL
LIN {X 0,Y 139.414,Z 416.221,A -85,B 0,C 180,E1 -25893.018,E2 -25893.018} C_VEL
LIN {X 0,Y 137.134,Z 421.092,A -85,B 0,C 180,E1 -25894.379,E2 -25894.379} C_VEL
LIN {X 0,Y 135.121,Z 423.983,A -85,B 0,C 180,E1 -25895.82,E2 -25895.82} C_VEL
LIN {X 0,Y 131.93,Z 433.651,A -85,B 0,C 180,E1 -25897.074,E2 -25897.074} C_VEL
LIN {X 0,Y 129.039,Z 439.93,A -85,B 0,C 180,E1 -25898.398,E2 -25898.398} C_VEL
LIN {X 0,Y 126.395,Z 444.295,A -85,B 0,C 180,E1 -25899.916,E2 -25899.916} C_VEL
LIN {X 0,Y 124.084,Z 446.92,A -85,B 0,C 180,E1 -25901.849,E2 -25901.849} C_VEL
LIN {X 0,Y 122.616,Z 448.3,A -85,B 0,C 180,E1 -25903.346,E2 -25903.346} C_VEL
LIN {X 0,Y 120.238,Z 452.44,A -85,B 0,C 180,E1 -25904.75,E2 -25904.75} C_VEL
LIN {X 0,Y 118.32,Z 455.244,A -85,B 0,C 180,E1 -25906.255,E2 -25906.255} C_VEL
LIN {X 0,Y 117.054,Z 456.597,A -85,B 0,C 180,E1 -25907.869,E2 -25907.869} C_VEL
LIN {X 0,Y 116.801,Z 456.412,A -85,B 0,C 180,E1 -25908.723,E2 -25908.723} C_VEL
LIN {X 0,Y 117.022,Z 455.278,A -85,B 0,C 180,E1 -25909.401,E2 -25909.401} C_VEL
LIN {X 0,Y 117.121,Z 454.934,A -85,B 0,C 180,E1 -25909.52,E2 -25909.52} C_VEL
LIN {X 0,Y 116.533,Z 468.011,A -85,B 0,C 180,E1 -25913.507,E2 -25913.507} C_VEL
LIN {X 0,Y 116.192,Z 478.24,A -85,B 0,C 180,E1 -25917.4,E2 -25917.4} C_VEL
LIN {X 0,Y 116.125,Z 489.339,A -85,B 0,C 180,E1 -25922.601,E2 -25922.601} C_VEL
LIN {X 0,Y 116.274,Z 498.153,A -85,B 0,C 180,E1 -25927.816,E2 -25927.816} C_VEL
LIN {X 0,Y 117.019,Z 505.418,A -85,B 0,C 180,E1 -25933.016,E2 -25933.016} C_VEL
LIN {X 0,Y 119.382,Z 512.909,A -85,B 0,C 180,E1 -25939.204,E2 -25939.204} C_VEL
LIN {X 0,Y 123.461,Z 519.295,A -85,B 0,C 180,E1 -25945.273,E2 -25945.273} C_VEL
LIN {X 0,Y 129.382,Z 524.651,A -85,B 0,C 180,E1 -25951.067,E2 -25951.067} C_VEL
LIN {X 0,Y 134.939,Z 527.923,A -85,B 0,C 180,E1 -25954.953,E2 -25954.953} C_VEL
LIN {X 0,Y 143.547,Z 531.234,A -85,B 0,C 180,E1 -25959.529,E2 -25959.529} C_VEL
LIN {X 0,Y 152.083,Z 533.213,A -85,B 0,C 180,E1 -25962.951,E2 -25962.951} C_VEL
LIN {X 0,Y 152.199,Z 533.389,A -85,B 0,C 180,E1 -25963.82,E2 -25963.82} C_VEL
LIN {X 0,Y 143.134,Z 532.545,A -85,B 0,C 180,E1 -25967.435,E2 -25967.435} C_VEL
LIN {X 0,Y 135.561,Z 530.993,A -85,B 0,C 180,E1 -25971.525,E2 -25971.525} C_VEL
LIN {X 0,Y 128.386,Z 528.35,A -85,B 0,C 180,E1 -25976.807,E2 -25976.807} C_VEL
LIN {X 0,Y 122.771,Z 524.651,A -85,B 0,C 180,E1 -25982.856,E2 -25982.856} C_VEL
LIN {X 0,Y 118.599,Z 529.296,A -85,B 0,C 180,E1 -25987.342,E2 -25987.342} C_VEL
LIN {X 0,Y 115.55,Z 532.948,A -85,B 0,C 180,E1 -25992.292,E2 -25992.292} C_VEL
LIN {X 0,Y 114.112,Z 534.837,A -85,B 0,C 180,E1 -25995.735,E2 -25995.735} C_VEL
LIN {X 0,Y 113.136,Z 536.265,A -85,B 0,C 180,E1 -25999.256,E2 -25999.256} C_VEL
LIN {X 0,Y 112.608,Z 537.281,A -85,B 0,C 180,E1 -26002.826,E2 -26002.826} C_VEL
LIN {X 0,Y 112.481,Z 538.075,A -85,B 0,C 180,E1 -26008.611,E2 -26008.611} C_VEL
LIN {X 0,Y 112.471,Z 538.079,A -85,B 0,C 180,E1 -26011.165,E2 -26011.165} C_VEL
LIN {X 0,Y 112.332,Z 537.241,A -85,B 0,C 180,E1 -26017.185,E2 -26017.185} C_VEL
LIN {X 0,Y 112.708,Z 536.207,A -85,B 0,C 180,E1 -26020.778,E2 -26020.778} C_VEL
LIN {X 0,Y 113.407,Z 534.743,A -85,B 0,C 180,E1 -26024.349,E2 -26024.349} C_VEL
LIN {X 0,Y 115.225,Z 531.73,A -85,B 0,C 180,E1 -26029.597,E2 -26029.597} C_VEL
LIN {X 0,Y 118.563,Z 526.896,A -85,B 0,C 180,E1 -26035.4,E2 -26035.4} C_VEL
LIN {X 0,Y 122.36,Z 521.406,A -85,B 0,C 180,E1 -26040.166,E2 -26040.166} C_VEL
LIN {X 0,Y 126.837,Z 514.591,A -85,B 0,C 180,E1 -26044.603,E2 -26044.603} C_VEL
LIN {X 0,Y 129.13,Z 510.958,A -85,B 0,C 180,E1 -26046.508,E2 -26046.508} C_VEL
LIN {X 0,Y 130.921,Z 507.288,A -85,B 0,C 180,E1 -26048.393,E2 -26048.393} C_VEL
LIN {X 0,Y 132.471,Z 500.928,A -85,B 0,C 180,E1 -26051.637,E2 -26051.637} C_VEL
LIN {X 0,Y 134.092,Z 493.997,A -85,B 0,C 180,E1 -26054.601,E2 -26054.601} C_VEL
LIN {X 0,Y 135.899,Z 489.434,A -85,B 0,C 180,E1 -26055.995,E2 -26055.995} C_VEL
LIN {X 0,Y 140.986,Z 478.359,A -85,B 0,C 180,E1 -26058.39,E2 -26058.39} C_VEL
LIN {X 0,Y 145.275,Z 467.153,A -85,B 0,C 180,E1 -26060.169,E2 -26060.169} C_VEL
LIN {X 0,Y 149.067,Z 454.39,A -85,B 0,C 180,E1 -26061.606,E2 -26061.606} C_VEL
LIN {X 0,Y 151.89,Z 441.345,A -85,B 0,C 180,E1 -26062.595,E2 -26062.595} C_VEL
LIN {X 0,Y 153.486,Z 428.402,A -85,B 0,C 180,E1 -26063.24,E2 -26063.24} C_VEL
LIN {X 0,Y 155.682,Z 400.709,A -85,B 0,C 180,E1 -26064.262,E2 -26064.262} C_VEL
LIN {X 0,Y 155.461,Z 395.385,A -85,B 0,C 180,E1 -26064.788,E2 -26064.788} C_VEL
LIN {X 0,Y 150.946,Z 386.453,A -85,B 0,C 180,E1 -26068.045,E2 -26068.045} C_VEL
LIN {X 0,Y 146.046,Z 377.776,A -85,B 0,C 180,E1 -26072.116,E2 -26072.116} C_VEL
LIN {X 0,Y 142.994,Z 373.091,A -85,B 0,C 180,E1 -26075.035,E2 -26075.035} C_VEL
LIN {X 0,Y 140.933,Z 369.962,A -85,B 0,C 180,E1 -26077.277,E2 -26077.277} C_VEL
LIN {X 0,Y 138.342,Z 366.173,A -85,B 0,C 180,E1 -26080.526,E2 -26080.526} C_VEL
LIN {X 0,Y 135.919,Z 362.72,A -85,B 0,C 180,E1 -26084.249,E2 -26084.249} C_VEL
LIN {X 0,Y 135.344,Z 361.651,A -85,B 0,C 180,E1 -26085.336,E2 -26085.336} C_VEL
LIN {X 0,Y 133.002,Z 359.019,A -85,B 0,C 180,E1 -26090.579,E2 -26090.579} C_VEL
LIN {X 0,Y 132.236,Z 356.499,A -85,B 0,C 180,E1 -26093.898,E2 -26093.898} C_VEL
LIN {X 0,Y 131.497,Z 355.978,A -85,B 0,C 180,E1 -26100,E2 -26100} C_VEL
LIN {X 0,Y 132.254,Z 356.633,A -85,B 0,C 180,E1 -26106.676,E2 -26106.676} C_VEL
LIN {X 0,Y 133.421,Z 359.829,A -85,B 0,C 180,E1 -26111.104,E2 -26111.104} C_VEL
LIN {X 0,Y 135.652,Z 362.116,A -85,B 0,C 180,E1 -26115.687,E2 -26115.687} C_VEL
LIN {X 0,Y 137.884,Z 365.693,A -85,B 0,C 180,E1 -26119.313,E2 -26119.313} C_VEL
LIN {X 0,Y 138.953,Z 366.977,A -85,B 0,C 180,E1 -26120.735,E2 -26120.735} C_VEL
LIN {X 0,Y 142.021,Z 371.58,A -85,B 0,C 180,E1 -26124.387,E2 -26124.387} C_VEL
LIN {X 0,Y 144.703,Z 375.784,A -85,B 0,C 180,E1 -26127.112,E2 -26127.112} C_VEL
LIN {X 0,Y 148.259,Z 381.631,A -85,B 0,C 180,E1 -26130.267,E2 -26130.267} C_VEL
LIN {X 0,Y 153.105,Z 390.614,A -85,B 0,C 180,E1 -26134.018,E2 -26134.018} C_VEL
LIN {X 0,Y 156.231,Z 397.056,A -85,B 0,C 180,E1 -26136.193,E2 -26136.193} C_VEL
LIN {X 0,Y 153.835,Z 425.938,A -85,B 0,C 180,E1 -26137.32,E2 -26137.32} C_VEL
LIN {X 0,Y 151.907,Z 438.489,A -85,B 0,C 180,E1 -26138.144,E2 -26138.144} C_VEL
LIN {X 0,Y 148.92,Z 451.178,A -85,B 0,C 180,E1 -26139.4,E2 -26139.4} C_VEL
LIN {X 0,Y 145.451,Z 462.498,A -85,B 0,C 180,E1 -26140.981,E2 -26140.981} C_VEL
LIN {X 0,Y 141.379,Z 472.881,A -85,B 0,C 180,E1 -26142.847,E2 -26142.847} C_VEL
LIN {X 0,Y 136.406,Z 483.504,A -85,B 0,C 180,E1 -26145.417,E2 -26145.417} C_VEL
LIN {X 0,Y 131.454,Z 492.821,A -85,B 0,C 180,E1 -26148.46,E2 -26148.46} C_VEL
LIN {X 0,Y 126.145,Z 501.549,A -85,B 0,C 180,E1 -26152.209,E2 -26152.209} C_VEL
LIN {X 0,Y 120.843,Z 509.011,A -85,B 0,C 180,E1 -26156.465,E2 -26156.465} C_VEL
LIN {X 0,Y 116.332,Z 514.991,A -85,B 0,C 180,E1 -26161.103,E2 -26161.103} C_VEL
LIN {X 0,Y 112.532,Z 519.712,A -85,B 0,C 180,E1 -26166.054,E2 -26166.054} C_VEL
LIN {X 0,Y 109.58,Z 523.312,A -85,B 0,C 180,E1 -26171.3,E2 -26171.3} C_VEL
LIN {X 0,Y 108.056,Z 525.164,A -85,B 0,C 180,E1 -26174.924,E2 -26174.924} C_VEL
LIN {X 0,Y 106.919,Z 526.571,A -85,B 0,C 180,E1 -26178.631,E2 -26178.631} C_VEL
LIN {X 0,Y 105.654,Z 528.164,A -85,B 0,C 180,E1 -26186.19,E2 -26186.19} C_VEL
LIN {X 0,Y 105.509,Z 528.391,A -85,B 0,C 180,E1 -26190.004,E2 -26190.004} C_VEL
LIN {X 0,Y 105.655,Z 528.192,A -85,B 0,C 180,E1 -26193.818,E2 -26193.818} C_VEL
LIN {X 0,Y 106.88,Z 526.639,A -85,B 0,C 180,E1 -26201.381,E2 -26201.381} C_VEL
LIN {X 0,Y 108.02,Z 525.269,A -85,B 0,C 180,E1 -26205.088,E2 -26205.088} C_VEL
LIN {X 0,Y 110.417,Z 522.392,A -85,B 0,C 180,E1 -26210.495,E2 -26210.495} C_VEL
LIN {X 0,Y 113.661,Z 518.474,A -85,B 0,C 180,E1 -26215.651,E2 -26215.651} C_VEL
LIN {X 0,Y 117.688,Z 513.393,A -85,B 0,C 180,E1 -26220.508,E2 -26220.508} C_VEL
LIN {X 0,Y 122.486,Z 506.982,A -85,B 0,C 180,E1 -26225.018,E2 -26225.018} C_VEL
LIN {X 0,Y 127.993,Z 498.991,A -85,B 0,C 180,E1 -26229.161,E2 -26229.161} C_VEL
LIN {X 0,Y 133.07,Z 490.226,A -85,B 0,C 180,E1 -26232.67,E2 -26232.67} C_VEL
LIN {X 0,Y 137.995,Z 480.731,A -85,B 0,C 180,E1 -26235.484,E2 -26235.484} C_VEL
LIN {X 0,Y 143.071,Z 469.371,A -85,B 0,C 180,E1 -26237.989,E2 -26237.989} C_VEL
LIN {X 0,Y 147.099,Z 458.099,A -85,B 0,C 180,E1 -26239.861,E2 -26239.861} C_VEL
LIN {X 0,Y 150.387,Z 446.503,A -85,B 0,C 180,E1 -26241.251,E2 -26241.251} C_VEL
LIN {X 0,Y 153.015,Z 433.41,A -85,B 0,C 180,E1 -26242.389,E2 -26242.389} C_VEL
LIN {X 0,Y 154.69,Z 419.979,A -85,B 0,C 180,E1 -26243.081,E2 -26243.081} C_VEL
LIN {X 0,Y 156.498,Z 397.404,A -85,B 0,C 180,E1 -26243.906,E2 -26243.906} C_VEL
LIN {X 0,Y 153.62,Z 391.41,A -85,B 0,C 180,E1 -26245.906,E2 -26245.906} C_VEL
LIN {X 0,Y 152.622,Z 391.548,A -85,B 0,C 180,E1 -26246.456,E2 -26246.456} C_VEL
LIN {X 0,Y 149.719,Z 396.213,A -85,B 0,C 180,E1 -26247.767,E2 -26247.767} C_VEL
LIN {X 0,Y 145.278,Z 410.715,A -85,B 0,C 180,E1 -26249.271,E2 -26249.271} C_VEL
LIN {X 0,Y 141.77,Z 420.082,A -85,B 0,C 180,E1 -26250.791,E2 -26250.791} C_VEL
LIN {X 0,Y 138.849,Z 425.824,A -85,B 0,C 180,E1 -26252.287,E2 -26252.287} C_VEL
LIN {X 0,Y 136.802,Z 428.925,A -85,B 0,C 180,E1 -26253.493,E2 -26253.493} C_VEL
LIN {X 0,Y 133.648,Z 437.028,A -85,B 0,C 180,E1 -26254.497,E2 -26254.497} C_VEL
LIN {X 0,Y 130.454,Z 443.316,A -85,B 0,C 180,E1 -26255.689,E2 -26255.689} C_VEL
LIN {X 0,Y 127.156,Z 448.369,A -85,B 0,C 180,E1 -26257.238,E2 -26257.238} C_VEL
LIN {X 0,Y 125.265,Z 450.7,A -85,B 0,C 180,E1 -26258.397,E2 -26258.397} C_VEL
LIN {X 0,Y 122.336,Z 453.416,A -85,B 0,C 180,E1 -26260.711,E2 -26260.711} C_VEL
LIN {X 0,Y 117.614,Z 459.807,A -85,B 0,C 180,E1 -26263.599,E2 -26263.599} C_VEL
LIN {X 0,Y 116.893,Z 460.68,A -85,B 0,C 180,E1 -26264.16,E2 -26264.16} C_VEL
LIN {X 0,Y 115.277,Z 462.213,A -85,B 0,C 180,E1 -26265.885,E2 -26265.885} C_VEL
LIN {X 0,Y 113.54,Z 463.562,A -85,B 0,C 180,E1 -26268.394,E2 -26268.394} C_VEL
LIN {X 0,Y 111.576,Z 466.309,A -85,B 0,C 180,E1 -26270.025,E2 -26270.025} C_VEL
LIN {X 0,Y 110.783,Z 467.344,A -85,B 0,C 180,E1 -26270.874,E2 -26270.874} C_VEL
LIN {X 0,Y 109.68,Z 468.558,A -85,B 0,C 180,E1 -26272.637,E2 -26272.637} C_VEL
LIN {X 0,Y 109.518,Z 468.294,A -85,B 0,C 180,E1 -26274.476,E2 -26274.476} C_VEL
LIN {X 0,Y 109.864,Z 467.571,A -85,B 0,C 180,E1 -26274.954,E2 -26274.954} C_VEL
LIN {X 0,Y 109.651,Z 477.805,A -85,B 0,C 180,E1 -26279.082,E2 -26279.082} C_VEL
LIN {X 0,Y 109.732,Z 487.141,A -85,B 0,C 180,E1 -26283.672,E2 -26283.672} C_VEL
LIN {X 0,Y 109.996,Z 496.18,A -85,B 0,C 180,E1 -26289.191,E2 -26289.191} C_VEL
LIN {X 0,Y 111.17,Z 504.79,A -85,B 0,C 180,E1 -26295.586,E2 -26295.586} C_VEL
LIN {X 0,Y 114.429,Z 513.068,A -85,B 0,C 180,E1 -26302.683,E2 -26302.683} C_VEL
LIN {X 0,Y 120.224,Z 520.308,A -85,B 0,C 180,E1 -26309.794,E2 -26309.794} C_VEL
LIN {X 0,Y 127.278,Z 525.526,A -85,B 0,C 180,E1 -26315.436,E2 -26315.436} C_VEL
LIN {X 0,Y 133.562,Z 528.694,A -85,B 0,C 180,E1 -26319.156,E2 -26319.156} C_VEL
LIN {X 0,Y 141.866,Z 531.595,A -85,B 0,C 180,E1 -26322.929,E2 -26322.929} C_VEL
LIN {X 0,Y 142.349,Z 531.839,A -85,B 0,C 180,E1 -26323.713,E2 -26323.713} C_VEL
LIN {X 0,Y 134.498,Z 530.37,A -85,B 0,C 180,E1 -26327.208,E2 -26327.208} C_VEL
LIN {X 0,Y 126.328,Z 527.824,A -85,B 0,C 180,E1 -26332.265,E2 -26332.265} C_VEL
LIN {X 0,Y 119.674,Z 524.294,A -85,B 0,C 180,E1 -26338.09,E2 -26338.09} C_VEL
LIN {X 0,Y 117.842,Z 522.994,A -85,B 0,C 180,E1 -26340.154,E2 -26340.154} C_VEL
LIN {X 0,Y 113.39,Z 527.544,A -85,B 0,C 180,E1 -26344.283,E2 -26344.283} C_VEL
LIN {X 0,Y 109.76,Z 531.554,A -85,B 0,C 180,E1 -26349.376,E2 -26349.376} C_VEL
LIN {X 0,Y 107.237,Z 534.521,A -85,B 0,C 180,E1 -26354.799,E2 -26354.799} C_VEL
LIN {X 0,Y 106.167,Z 535.949,A -85,B 0,C 180,E1 -26358.542,E2 -26358.542} C_VEL
LIN {X 0,Y 105.335,Z 537.589,A -85,B 0,C 180,E1 -26366.171,E2 -26366.171} C_VEL
LIN {X 0,Y 105.426,Z 537.791,A -85,B 0,C 180,E1 -26370.619,E2 -26370.619} C_VEL
LIN {X 0,Y 105.269,Z 536.923,A -85,B 0,C 180,E1 -26377.669,E2 -26377.669} C_VEL
LIN {X 0,Y 105.693,Z 535.887,A -85,B 0,C 180,E1 -26381.503,E2 -26381.503} C_VEL
LIN {X 0,Y 106.497,Z 534.424,A -85,B 0,C 180,E1 -26385.302,E2 -26385.302} C_VEL
LIN {X 0,Y 108.528,Z 531.41,A -85,B 0,C 180,E1 -26390.861,E2 -26390.861} C_VEL
LIN {X 0,Y 111.579,Z 527.344,A -85,B 0,C 180,E1 -26396.157,E2 -26396.157} C_VEL
LIN {X 0,Y 115.545,Z 522.097,A -85,B 0,C 180,E1 -26401.128,E2 -26401.128} C_VEL
LIN {X 0,Y 120.19,Z 515.502,A -85,B 0,C 180,E1 -26405.78,E2 -26405.78} C_VEL
LIN {X 0,Y 125.651,Z 507.328,A -85,B 0,C 180,E1 -26410.028,E2 -26410.028} C_VEL
LIN {X 0,Y 130.758,Z 498.952,A -85,B 0,C 180,E1 -26413.254,E2 -26413.254} C_VEL
LIN {X 0,Y 135.899,Z 489.434,A -85,B 0,C 180,E1 -26415.995,E2 -26415.995} C_VEL
LIN {X 0,Y 137.658,Z 484.787,A -85,B 0,C 180,E1 -26417.299,E2 -26417.299} C_VEL
LIN {X 0,Y 139.15,Z 476.953,A -85,B 0,C 180,E1 -26419.743,E2 -26419.743} C_VEL
LIN {X 0,Y 140.525,Z 468.728,A -85,B 0,C 180,E1 -26421.936,E2 -26421.936} C_VEL
LIN {X 0,Y 142.014,Z 463.38,A -85,B 0,C 180,E1 -26422.818,E2 -26422.818} C_VEL
LIN {X 0,Y 145.432,Z 451.579,A -85,B 0,C 180,E1 -26424.036,E2 -26424.036} C_VEL
LIN {X 0,Y 148.121,Z 438.478,A -85,B 0,C 180,E1 -26424.92,E2 -26424.92} C_VEL
LIN {X 0,Y 149.781,Z 423.091,A -85,B 0,C 180,E1 -26425.608,E2 -26425.608} C_VEL
LIN {X 0,Y 151.56,Z 401.323,A -85,B 0,C 180,E1 -26426.418,E2 -26426.418} C_VEL
LIN {X 0,Y 151.358,Z 398.74,A -85,B 0,C 180,E1 -26426.75,E2 -26426.75} C_VEL
LIN {X 0,Y 147.098,Z 390.106,A -85,B 0,C 180,E1 -26430.161,E2 -26430.161} C_VEL
LIN {X 0,Y 142.995,Z 382.729,A -85,B 0,C 180,E1 -26433.943,E2 -26433.943} C_VEL
LIN {X 0,Y 139.458,Z 376.9,A -85,B 0,C 180,E1 -26437.817,E2 -26437.817} C_VEL
LIN {X 0,Y 136.714,Z 372.729,A -85,B 0,C 180,E1 -26441.453,E2 -26441.453} C_VEL
LIN {X 0,Y 134.35,Z 369.071,A -85,B 0,C 180,E1 -26445.419,E2 -26445.419} C_VEL
LIN {X 0,Y 133.794,Z 368.295,A -85,B 0,C 180,E1 -26446.521,E2 -26446.521} C_VEL
LIN {X 0,Y 131.81,Z 365.641,A -85,B 0,C 180,E1 -26451.569,E2 -26451.569} C_VEL
LIN {X 0,Y 131.203,Z 363.462,A -85,B 0,C 180,E1 -26454.621,E2 -26454.621} C_VEL
LIN {X 0,Y 130.65,Z 363.149,A -85,B 0,C 180,E1 -26461.541,E2 -26461.541} C_VEL
LIN {X 0,Y 131.286,Z 363.779,A -85,B 0,C 180,E1 -26466.339,E2 -26466.339} C_VEL
LIN {X 0,Y 132.445,Z 366.906,A -85,B 0,C 180,E1 -26470.897,E2 -26470.897} C_VEL
LIN {X 0,Y 134.213,Z 368.742,A -85,B 0,C 180,E1 -26474.742,E2 -26474.742} C_VEL
LIN {X 0,Y 136.376,Z 372.352,A -85,B 0,C 180,E1 -26478.518,E2 -26478.518} C_VEL
LIN {X 0,Y 137.433,Z 373.878,A -85,B 0,C 180,E1 -26480.039,E2 -26480.039} C_VEL
LIN {X 0,Y 140.214,Z 378.218,A -85,B 0,C 180,E1 -26483.542,E2 -26483.542} C_VEL
LIN {X 0,Y 143.798,Z 384.07,A -85,B 0,C 180,E1 -26487.297,E2 -26487.297} C_VEL
LIN {X 0,Y 148.407,Z 392.679,A -85,B 0,C 180,E1 -26491.394,E2 -26491.394} C_VEL
LIN {X 0,Y 151.953,Z 400.094,A -85,B 0,C 180,E1 -26494.159,E2 -26494.159} C_VEL
LIN {X 0,Y 149.513,Z 427.325,A -85,B 0,C 180,E1 -26495.214,E2 -26495.214} C_VEL
LIN {X 0,Y 147.325,Z 440.22,A -85,B 0,C 180,E1 -26496.106,E2 -26496.106} C_VEL
LIN {X 0,Y 144.21,Z 452.562,A -85,B 0,C 180,E1 -26497.352,E2 -26497.352} C_VEL
LIN {X 0,Y 140.912,Z 462.803,A -85,B 0,C 180,E1 -26498.809,E2 -26498.809} C_VEL
LIN {X 0,Y 136.652,Z 473.191,A -85,B 0,C 180,E1 -26500.665,E2 -26500.665} C_VEL
LIN {X 0,Y 131.463,Z 483.815,A -85,B 0,C 180,E1 -26503.253,E2 -26503.253} C_VEL
LIN {X 0,Y 126.016,Z 493.514,A -85,B 0,C 180,E1 -26506.471,E2 -26506.471} C_VEL
LIN {X 0,Y 120.622,Z 501.864,A -85,B 0,C 180,E1 -26510.145,E2 -26510.145} C_VEL
LIN {X 0,Y 115.007,Z 509.326,A -85,B 0,C 180,E1 -26514.516,E2 -26514.516} C_VEL
LIN {X 0,Y 110.161,Z 515.308,A -85,B 0,C 180,E1 -26519.315,E2 -26519.315} C_VEL
LIN {X 0,Y 106.089,Z 520.029,A -85,B 0,C 180,E1 -26524.499,E2 -26524.499} C_VEL
LIN {X 0,Y 102.873,Z 523.63,A -85,B 0,C 180,E1 -26530.031,E2 -26530.031} C_VEL
LIN {X 0,Y 101.224,Z 525.482,A -85,B 0,C 180,E1 -26533.88,E2 -26533.88} C_VEL
LIN {X 0,Y 99.98,Z 526.888,A -85,B 0,C 180,E1 -26537.83,E2 -26537.83} C_VEL
LIN {X 0,Y 98.585,Z 528.48,A -85,B 0,C 180,E1 -26545.916,E2 -26545.916} C_VEL
LIN {X 0,Y 98.444,Z 528.649,A -85,B 0,C 180,E1 -26551.845,E2 -26551.845} C_VEL
LIN {X 0,Y 99.076,Z 527.922,A -85,B 0,C 180,E1 -26558.16,E2 -26558.16} C_VEL
LIN {X 0,Y 99.926,Z 526.955,A -85,B 0,C 180,E1 -26562.185,E2 -26562.185} C_VEL
LIN {X 0,Y 101.193,Z 525.585,A -85,B 0,C 180,E1 -26566.133,E2 -26566.133} C_VEL
LIN {X 0,Y 103.798,Z 522.708,A -85,B 0,C 180,E1 -26571.868,E2 -26571.868} C_VEL
LIN {X 0,Y 107.314,Z 518.788,A -85,B 0,C 180,E1 -26577.29,E2 -26577.29} C_VEL
LIN {X 0,Y 111.631,Z 513.707,A -85,B 0,C 180,E1 -26582.357,E2 -26582.357} C_VEL
LIN {X 0,Y 116.751,Z 507.294,A -85,B 0,C 180,E1 -26587.015,E2 -26587.015} C_VEL
LIN {X 0,Y 122.571,Z 499.302,A -85,B 0,C 180,E1 -26591.257,E2 -26591.257} C_VEL
LIN {X 0,Y 128.068,Z 490.305,A -85,B 0,C 180,E1 -26594.903,E2 -26594.903} C_VEL
LIN {X 0,Y 133.714,Z 479.891,A -85,B 0,C 180,E1 -26597.941,E2 -26597.941} C_VEL
LIN {X 0,Y 138.435,Z 469.67,A -85,B 0,C 180,E1 -26600.166,E2 -26600.166} C_VEL
LIN {X 0,Y 142.635,Z 458.389,A -85,B 0,C 180,E1 -26602.037,E2 -26602.037} C_VEL
LIN {X 0,Y 146.354,Z 445.542,A -85,B 0,C 180,E1 -26603.551,E2 -26603.551} C_VEL
LIN {X 0,Y 148.888,Z 433.164,A -85,B 0,C 180,E1 -26604.586,E2 -26604.586} C_VEL
LIN {X 0,Y 150.628,Z 419.273,A -85,B 0,C 180,E1 -26605.267,E2 -26605.267} C_VEL
LIN {X 0,Y 152.06,Z 402.112,A -85,B 0,C 180,E1 -26605.891,E2 -26605.891} C_VEL
LIN {X 0,Y 147.723,Z 415.446,A -85,B 0,C 180,E1 -26607.278,E2 -26607.278} C_VEL
LIN {X 0,Y 143.952,Z 424.598,A -85,B 0,C 180,E1 -26608.752,E2 -26608.752} C_VEL
LIN {X 0,Y 140.41,Z 430.793,A -85,B 0,C 180,E1 -26610.305,E2 -26610.305} C_VEL
LIN {X 0,Y 138.75,Z 433.188,A -85,B 0,C 180,E1 -26611.117,E2 -26611.117} C_VEL
LIN {X 0,Y 134.902,Z 441.69,A -85,B 0,C 180,E1 -26612.144,E2 -26612.144} C_VEL
LIN {X 0,Y 130.926,Z 448.41,A -85,B 0,C 180,E1 -26613.439,E2 -26613.439} C_VEL
LIN {X 0,Y 127.288,Z 453.28,A -85,B 0,C 180,E1 -26614.939,E2 -26614.939} C_VEL
LIN {X 0,Y 124.154,Z 456.603,A -85,B 0,C 180,E1 -26616.656,E2 -26616.656} C_VEL
LIN {X 0,Y 121.938,Z 458.497,A -85,B 0,C 180,E1 -26618.176,E2 -26618.176} C_VEL
LIN {X 0,Y 116.091,Z 465.222,A -85,B 0,C 180,E1 -26621.468,E2 -26621.468} C_VEL
LIN {X 0,Y 115.059,Z 466.28,A -85,B 0,C 180,E1 -26622.217,E2 -26622.217} C_VEL
LIN {X 0,Y 113.489,Z 467.57,A -85,B 0,C 180,E1 -26623.672,E2 -26623.672} C_VEL
LIN {X 0,Y 111.965,Z 468.667,A -85,B 0,C 180,E1 -26625.458,E2 -26625.458} C_VEL
LIN {X 0,Y 108.3,Z 472.646,A -85,B 0,C 180,E1 -26628.774,E2 -26628.774} C_VEL
LIN {X 0,Y 106.781,Z 474.092,A -85,B 0,C 180,E1 -26630.863,E2 -26630.863} C_VEL
LIN {X 0,Y 105.362,Z 475.303,A -85,B 0,C 180,E1 -26634.257,E2 -26634.257} C_VEL
LIN {X 0,Y 103.876,Z 477.322,A -85,B 0,C 180,E1 -26636.12,E2 -26636.12} C_VEL
LIN {X 0,Y 102.574,Z 479.155,A -85,B 0,C 180,E1 -26640,E2 -26640} C_VEL
LIN {X 0,Y 102.81,Z 478.913,A -85,B 0,C 180,E1 -26640.979,E2 -26640.979} C_VEL
LIN {X 0,Y 103.248,Z 478.431,A -85,B 0,C 180,E1 -26641.584,E2 -26641.584} C_VEL
LIN {X 0,Y 103.47,Z 486.46,A -85,B 0,C 180,E1 -26645.848,E2 -26645.848} C_VEL
LIN {X 0,Y 103.956,Z 495.45,A -85,B 0,C 180,E1 -26651.702,E2 -26651.702} C_VEL
LIN {X 0,Y 105.56,Z 504.037,A -85,B 0,C 180,E1 -26658.436,E2 -26658.436} C_VEL
LIN {X 0,Y 109.005,Z 511.547,A -85,B 0,C 180,E1 -26665.012,E2 -26665.012} C_VEL
LIN {X 0,Y 114.393,Z 518.245,A -85,B 0,C 180,E1 -26671.481,E2 -26671.481} C_VEL
LIN {X 0,Y 121.706,Z 523.899,A -85,B 0,C 180,E1 -26677.325,E2 -26677.325} C_VEL
LIN {X 0,Y 128.234,Z 527.412,A -85,B 0,C 180,E1 -26681.123,E2 -26681.123} C_VEL
LIN {X 0,Y 133.002,Z 529.403,A -85,B 0,C 180,E1 -26683.388,E2 -26683.388} C_VEL
LIN {X 0,Y 125.139,Z 527.207,A -85,B 0,C 180,E1 -26687.624,E2 -26687.624} C_VEL
LIN {X 0,Y 115.683,Z 522.784,A -85,B 0,C 180,E1 -26694.746,E2 -26694.746} C_VEL
LIN {X 0,Y 113.245,Z 521.208,A -85,B 0,C 180,E1 -26697.238,E2 -26697.238} C_VEL
LIN {X 0,Y 108.672,Z 525.632,A -85,B 0,C 180,E1 -26700.981,E2 -26700.981} C_VEL
LIN {X 0,Y 104.346,Z 530.005,A -85,B 0,C 180,E1 -26706.16,E2 -26706.16} C_VEL
LIN {X 0,Y 102.099,Z 532.316,A -85,B 0,C 180,E1 -26709.864,E2 -26709.864} C_VEL
LIN {X 0,Y 100.405,Z 534.205,A -85,B 0,C 180,E1 -26713.736,E2 -26713.736} C_VEL
LIN {X 0,Y 99.203,Z 535.631,A -85,B 0,C 180,E1 -26717.725,E2 -26717.725} C_VEL
LIN {X 0,Y 98.247,Z 537.272,A -85,B 0,C 180,E1 -26725.894,E2 -26725.894} C_VEL
LIN {X 0,Y 98.392,Z 537.5,A -85,B 0,C 180,E1 -26729.996,E2 -26729.996} C_VEL
LIN {X 0,Y 98.134,Z 537.25,A -85,B 0,C 180,E1 -26734.103,E2 -26734.103} C_VEL
LIN {X 0,Y 98.709,Z 535.568,A -85,B 0,C 180,E1 -26742.329,E2 -26742.329} C_VEL
LIN {X 0,Y 99.629,Z 534.104,A -85,B 0,C 180,E1 -26746.385,E2 -26746.385} C_VEL
LIN {X 0,Y 101.894,Z 531.092,A -85,B 0,C 180,E1 -26752.289,E2 -26752.289} C_VEL
LIN {X 0,Y 105.216,Z 527.025,A -85,B 0,C 180,E1 -26757.872,E2 -26757.872} C_VEL
LIN {X 0,Y 109.791,Z 521.316,A -85,B 0,C 180,E1 -26763.459,E2 -26763.459} C_VEL
LIN {X 0,Y 115.361,Z 513.956,A -85,B 0,C 180,E1 -26768.637,E2 -26768.637} C_VEL
LIN {X 0,Y 121.306,Z 505.449,A -85,B 0,C 180,E1 -26772.897,E2 -26772.897} C_VEL
LIN {X 0,Y 126.781,Z 496.711,A -85,B 0,C 180,E1 -26776.103,E2 -26776.103} C_VEL
LIN {X 0,Y 132.69,Z 485.963,A -85,B 0,C 180,E1 -26778.999,E2 -26778.999} C_VEL
LIN {X 0,Y 137.623,Z 475.109,A -85,B 0,C 180,E1 -26781.143,E2 -26781.143} C_VEL
LIN {X 0,Y 142.014,Z 463.38,A -85,B 0,C 180,E1 -26782.818,E2 -26782.818} C_VEL
LIN {X 0,Y 143.373,Z 457.983,A -85,B 0,C 180,E1 -26783.627,E2 -26783.627} C_VEL
LIN {X 0,Y 144.072,Z 449.094,A -85,B 0,C 180,E1 -26785.38,E2 -26785.38} C_VEL
LIN {X 0,Y 144.258,Z 439.972,A -85,B 0,C 180,E1 -26786.951,E2 -26786.951} C_VEL
LIN {X 0,Y 144.738,Z 434.211,A -85,B 0,C 180,E1 -26787.456,E2 -26787.456} C_VEL
LIN {X 0,Y 147.616,Z 402.519,A -85,B 0,C 180,E1 -26788.669,E2 -26788.669} C_VEL
LIN {X 0,Y 143.473,Z 393.889,A -85,B 0,C 180,E1 -26792.366,E2 -26792.366} C_VEL
LIN {X 0,Y 139.606,Z 386.67,A -85,B 0,C 180,E1 -26796.421,E2 -26796.421} C_VEL
LIN {X 0,Y 137.063,Z 382.523,A -85,B 0,C 180,E1 -26799.555,E2 -26799.555} C_VEL
LIN {X 0,Y 135,Z 379.179,A -85,B 0,C 180,E1 -26802.582,E2 -26802.582} C_VEL
LIN {X 0,Y 132.659,Z 375.218,A -85,B 0,C 180,E1 -26806.988,E2 -26806.988} C_VEL
LIN {X 0,Y 130.726,Z 372.478,A -85,B 0,C 180,E1 -26812.276,E2 -26812.276} C_VEL
LIN {X 0,Y 130.189,Z 370.44,A -85,B 0,C 180,E1 -26815.356,E2 -26815.356} C_VEL
LIN {X 0,Y 129.785,Z 370.201,A -85,B 0,C 180,E1 -26821.552,E2 -26821.552} C_VEL
LIN {X 0,Y 130.297,Z 370.784,A -85,B 0,C 180,E1 -26825.805,E2 -26825.805} C_VEL
LIN {X 0,Y 131.37,Z 373.838,A -85,B 0,C 180,E1 -26830.402,E2 -26830.402} C_VEL
LIN {X 0,Y 132.976,Z 375.742,A -85,B 0,C 180,E1 -26834.149,E2 -26834.149} C_VEL
LIN {X 0,Y 135.278,Z 379.472,A -85,B 0,C 180,E1 -26838.29,E2 -26838.29} C_VEL
LIN {X 0,Y 138.37,Z 384.726,A -85,B 0,C 180,E1 -26842.589,E2 -26842.589} C_VEL
LIN {X 0,Y 141.296,Z 389.743,A -85,B 0,C 180,E1 -26845.899,E2 -26845.899} C_VEL
LIN {X 0,Y 145.594,Z 398.208,A -85,B 0,C 180,E1 -26850.054,E2 -26850.054} C_VEL
LIN {X 0,Y 147.843,Z 403.073,A -85,B 0,C 180,E1 -26851.984,E2 -26851.984} C_VEL
LIN {X 0,Y 145.483,Z 428.091,A -85,B 0,C 180,E1 -26852.966,E2 -26852.966} C_VEL
LIN {X 0,Y 143.115,Z 441.232,A -85,B 0,C 180,E1 -26853.884,E2 -26853.884} C_VEL
LIN {X 0,Y 139.696,Z 453.945,A -85,B 0,C 180,E1 -26855.168,E2 -26855.168} C_VEL
LIN {X 0,Y 135.944,Z 464.765,A -85,B 0,C 180,E1 -26856.75,E2 -26856.75} C_VEL
LIN {X 0,Y 130.926,Z 476.043,A -85,B 0,C 180,E1 -26858.896,E2 -26858.896} C_VEL
LIN {X 0,Y 125.546,Z 486.213,A -85,B 0,C 180,E1 -26861.525,E2 -26861.525} C_VEL
LIN {X 0,Y 120.738,Z 494.213,A -85,B 0,C 180,E1 -26864.307,E2 -26864.307} C_VEL
LIN {X 0,Y 115.259,Z 502.18,A -85,B 0,C 180,E1 -26867.881,E2 -26867.881} C_VEL
LIN {X 0,Y 109.321,Z 509.642,A -85,B 0,C 180,E1 -26872.363,E2 -26872.363} C_VEL
LIN {X 0,Y 104.11,Z 515.626,A -85,B 0,C 180,E1 -26877.318,E2 -26877.318} C_VEL
LIN {X 0,Y 99.739,Z 520.346,A -85,B 0,C 180,E1 -26882.746,E2 -26882.746} C_VEL
LIN {X 0,Y 96.233,Z 523.948,A -85,B 0,C 180,E1 -26888.588,E2 -26888.588} C_VEL
LIN {X 0,Y 94.441,Z 525.798,A -85,B 0,C 180,E1 -26892.687,E2 -26892.687} C_VEL
LIN {X 0,Y 93.052,Z 527.205,A -85,B 0,C 180,E1 -26896.909,E2 -26896.909} C_VEL
LIN {X 0,Y 91.52,Z 528.797,A -85,B 0,C 180,E1 -26905.6,E2 -26905.6} C_VEL
LIN {X 0,Y 91.365,Z 529.023,A -85,B 0,C 180,E1 -26910.004,E2 -26910.004} C_VEL
LIN {X 0,Y 91.521,Z 528.824,A -85,B 0,C 180,E1 -26914.409,E2 -26914.409} C_VEL
LIN {X 0,Y 93.014,Z 527.271,A -85,B 0,C 180,E1 -26923.106,E2 -26923.106} C_VEL
LIN {X 0,Y 94.392,Z 525.901,A -85,B 0,C 180,E1 -26927.331,E2 -26927.331} C_VEL
LIN {X 0,Y 97.252,Z 523.023,A -85,B 0,C 180,E1 -26933.424,E2 -26933.424} C_VEL
LIN {X 0,Y 101.071,Z 519.102,A -85,B 0,C 180,E1 -26939.131,E2 -26939.131} C_VEL
LIN {X 0,Y 105.708,Z 514.02,A -85,B 0,C 180,E1 -26944.415,E2 -26944.415} C_VEL
LIN {X 0,Y 111.174,Z 507.605,A -85,B 0,C 180,E1 -26949.214,E2 -26949.214} C_VEL
LIN {X 0,Y 117.326,Z 499.62,A -85,B 0,C 180,E1 -26953.538,E2 -26953.538} C_VEL
LIN {X 0,Y 123.146,Z 490.612,A -85,B 0,C 180,E1 -26957.233,E2 -26957.233} C_VEL
LIN {X 0,Y 129.076,Z 480.194,A -85,B 0,C 180,E1 -26960.276,E2 -26960.276} C_VEL
LIN {X 0,Y 134.005,Z 469.969,A -85,B 0,C 180,E1 -26962.494,E2 -26962.494} C_VEL
LIN {X 0,Y 138.392,Z 458.679,A -85,B 0,C 180,E1 -26964.349,E2 -26964.349} C_VEL
LIN {X 0,Y 142.259,Z 445.82,A -85,B 0,C 180,E1 -26965.847,E2 -26965.847} C_VEL
LIN {X 0,Y 144.955,Z 433.117,A -85,B 0,C 180,E1 -26966.887,E2 -26966.887} C_VEL
LIN {X 0,Y 145.268,Z 430.681,A -85,B 0,C 180,E1 -26967.069,E2 -26967.069} C_VEL
LIN {X 0,Y 141.315,Z 436.505,A -85,B 0,C 180,E1 -26968.591,E2 -26968.591} C_VEL
LIN {X 0,Y 140.588,Z 437.802,A -85,B 0,C 180,E1 -26968.824,E2 -26968.824} C_VEL
LIN {X 0,Y 135.761,Z 446.982,A -85,B 0,C 180,E1 -26969.922,E2 -26969.922} C_VEL
LIN {X 0,Y 131.31,Z 453.479,A -85,B 0,C 180,E1 -26971.203,E2 -26971.203} C_VEL
LIN {X 0,Y 126.773,Z 458.799,A -85,B 0,C 180,E1 -26972.873,E2 -26972.873} C_VEL
LIN {X 0,Y 123.161,Z 462.143,A -85,B 0,C 180,E1 -26974.661,E2 -26974.661} C_VEL
LIN {X 0,Y 120.963,Z 463.86,A -85,B 0,C 180,E1 -26976.002,E2 -26976.002} C_VEL
LIN {X 0,Y 115.574,Z 469.433,A -85,B 0,C 180,E1 -26978.601,E2 -26978.601} C_VEL
LIN {X 0,Y 113.234,Z 471.58,A -85,B 0,C 180,E1 -26980.04,E2 -26980.04} C_VEL
LIN {X 0,Y 109.872,Z 473.948,A -85,B 0,C 180,E1 -26983.079,E2 -26983.079} C_VEL
LIN {X 0,Y 107.798,Z 475.773,A -85,B 0,C 180,E1 -26984.883,E2 -26984.883} C_VEL
LIN {X 0,Y 105.712,Z 477.769,A -85,B 0,C 180,E1 -26986.544,E2 -26986.544} C_VEL
LIN {X 0,Y 104.203,Z 479.015,A -85,B 0,C 180,E1 -26988.326,E2 -26988.326} C_VEL
LIN {X 0,Y 102.097,Z 480.64,A -85,B 0,C 180,E1 -26992.087,E2 -26992.087} C_VEL
LIN {X 0,Y 100.573,Z 482.306,A -85,B 0,C 180,E1 -26993.983,E2 -26993.983} C_VEL
LIN {X 0,Y 99.581,Z 483.355,A -85,B 0,C 180,E1 -26995.953,E2 -26995.953} C_VEL
LIN {X 0,Y 98.398,Z 484.879,A -85,B 0,C 180,E1 -27000,E2 -27000} C_VEL
LIN {X 0,Y 98.413,Z 484.953,A -85,B 0,C 180,E1 -27001.002,E2 -27001.002} C_VEL
LIN {X 0,Y 96.906,Z 487.406,A -85,B 0,C 180,E1 -27004.159,E2 -27004.159} C_VEL
LIN {X 0,Y 96.564,Z 489.042,A -85,B 0,C 180,E1 -27008.37,E2 -27008.37} C_VEL
LIN {X 0,Y 97.166,Z 488.933,A -85,B 0,C 180,E1 -27009.891,E2 -27009.891} C_VEL
LIN {X 0,Y 97.574,Z 488.763,A -85,B 0,C 180,E1 -27010.374,E2 -27010.374} C_VEL
LIN {X 0,Y 98.596,Z 497.128,A -85,B 0,C 180,E1 -27016.566,E2 -27016.566} C_VEL
LIN {X 0,Y 101.774,Z 506.463,A -85,B 0,C 180,E1 -27024.477,E2 -27024.477} C_VEL
LIN {X 0,Y 107.092,Z 514.201,A -85,B 0,C 180,E1 -27031.669,E2 -27031.669} C_VEL
LIN {X 0,Y 114.268,Z 520.59,A -85,B 0,C 180,E1 -27037.955,E2 -27037.955} C_VEL
LIN {X 0,Y 123.093,Z 525.856,A -85,B 0,C 180,E1 -27043.247,E2 -27043.247} C_VEL
LIN {X 0,Y 120.269,Z 524.95,A -85,B 0,C 180,E1 -27045.47,E2 -27045.47} C_VEL
LIN {X 0,Y 112.164,Z 521.16,A -85,B 0,C 180,E1 -27051.197,E2 -27051.197} C_VEL
LIN {X 0,Y 109.127,Z 519.258,A -85,B 0,C 180,E1 -27054.004,E2 -27054.004} C_VEL
LIN {X 0,Y 104.366,Z 523.596,A -85,B 0,C 180,E1 -27057.399,E2 -27057.399} C_VEL
LIN {X 0,Y 99.292,Z 528.351,A -85,B 0,C 180,E1 -27062.604,E2 -27062.604} C_VEL
LIN {X 0,Y 95.454,Z 531.999,A -85,B 0,C 180,E1 -27068.395,E2 -27068.395} C_VEL
LIN {X 0,Y 93.617,Z 533.889,A -85,B 0,C 180,E1 -27072.521,E2 -27072.521} C_VEL
LIN {X 0,Y 92.274,Z 535.315,A -85,B 0,C 180,E1 -27076.787,E2 -27076.787} C_VEL
LIN {X 0,Y 91.171,Z 536.955,A -85,B 0,C 180,E1 -27085.574,E2 -27085.574} C_VEL
LIN {X 0,Y 91.285,Z 537.182,A -85,B 0,C 180,E1 -27089.996,E2 -27089.996} C_VEL
LIN {X 0,Y 91.051,Z 536.932,A -85,B 0,C 180,E1 -27094.422,E2 -27094.422} C_VEL
LIN {X 0,Y 91.76,Z 535.249,A -85,B 0,C 180,E1 -27103.279,E2 -27103.279} C_VEL
LIN {X 0,Y 92.792,Z 533.785,A -85,B 0,C 180,E1 -27107.631,E2 -27107.631} C_VEL
LIN {X 0,Y 95.335,Z 530.773,A -85,B 0,C 180,E1 -27113.915,E2 -27113.915} C_VEL
LIN {X 0,Y 98.966,Z 526.706,A -85,B 0,C 180,E1 -27119.803,E2 -27119.803} C_VEL
LIN {X 0,Y 103.437,Z 521.554,A -85,B 0,C 180,E1 -27125.157,E2 -27125.157} C_VEL
LIN {X 0,Y 108.91,Z 514.865,A -85,B 0,C 180,E1 -27130.183,E2 -27130.183} C_VEL
LIN {X 0,Y 115.083,Z 506.694,A -85,B 0,C 180,E1 -27134.606,E2 -27134.606} C_VEL
LIN {X 0,Y 120.77,Z 498.322,A -85,B 0,C 180,E1 -27137.894,E2 -27137.894} C_VEL
LIN {X 0,Y 126.888,Z 487.973,A -85,B 0,C 180,E1 -27140.838,E2 -27140.838} C_VEL
LIN {X 0,Y 132.626,Z 476.333,A -85,B 0,C 180,E1 -27143.267,E2 -27143.267} C_VEL
LIN {X 0,Y 137.281,Z 464.632,A -85,B 0,C 180,E1 -27144.99,E2 -27144.99} C_VEL
LIN {X 0,Y 141.037,Z 452.542,A -85,B 0,C 180,E1 -27146.253,E2 -27146.253} C_VEL
LIN {X 0,Y 143.962,Z 439.456,A -85,B 0,C 180,E1 -27147.163,E2 -27147.163} C_VEL
LIN {X 0,Y 144.738,Z 434.211,A -85,B 0,C 180,E1 -27147.456,E2 -27147.456} C_VEL
LIN {X 0,Y 144.849,Z 430.35,A -85,B 0,C 180,E1 -27147.842,E2 -27147.842} C_VEL
LIN {X 0,Y 142.984,Z 418.394,A -85,B 0,C 180,E1 -27150.241,E2 -27150.241} C_VEL
LIN {X 0,Y 142.997,Z 414.514,A -85,B 0,C 180,E1 -27150.609,E2 -27150.609} C_VEL
LIN {X 0,Y 143.763,Z 405.808,A -85,B 0,C 180,E1 -27150.935,E2 -27150.935} C_VEL
LIN {X 0,Y 140.126,Z 397.909,A -85,B 0,C 180,E1 -27154.607,E2 -27154.607} C_VEL
LIN {X 0,Y 136.948,Z 391.808,A -85,B 0,C 180,E1 -27158.365,E2 -27158.365} C_VEL
LIN {X 0,Y 135.118,Z 388.634,A -85,B 0,C 180,E1 -27160.881,E2 -27160.881} C_VEL
LIN {X 0,Y 133.399,Z 385.651,A -85,B 0,C 180,E1 -27163.649,E2 -27163.649} C_VEL
LIN {X 0,Y 131.447,Z 382.067,A -85,B 0,C 180,E1 -27167.651,E2 -27167.651} C_VEL
LIN {X 0,Y 129.623,Z 379.177,A -85,B 0,C 180,E1 -27173.189,E2 -27173.189} C_VEL
LIN {X 0,Y 129.259,Z 377.45,A -85,B 0,C 180,E1 -27175.713,E2 -27175.713} C_VEL
LIN {X 0,Y 128.919,Z 377.252,A -85,B 0,C 180,E1 -27181.562,E2 -27181.562} C_VEL
LIN {X 0,Y 129.297,Z 377.656,A -85,B 0,C 180,E1 -27185.068,E2 -27185.068} C_VEL
LIN {X 0,Y 130.368,Z 380.864,A -85,B 0,C 180,E1 -27190.091,E2 -27190.091} C_VEL
LIN {X 0,Y 131.655,Z 382.513,A -85,B 0,C 180,E1 -27193.31,E2 -27193.31} C_VEL
LIN {X 0,Y 134.124,Z 386.866,A -85,B 0,C 180,E1 -27198.028,E2 -27198.028} C_VEL
LIN {X 0,Y 136.371,Z 390.85,A -85,B 0,C 180,E1 -27201.345,E2 -27201.345} C_VEL
LIN {X 0,Y 139.13,Z 395.919,A -85,B 0,C 180,E1 -27204.74,E2 -27204.74} C_VEL
LIN {X 0,Y 143.048,Z 404.193,A -85,B 0,C 180,E1 -27208.845,E2 -27208.845} C_VEL
LIN {X 0,Y 143.963,Z 406.328,A -85,B 0,C 180,E1 -27209.719,E2 -27209.719} C_VEL
LIN {X 0,Y 141.738,Z 428.42,A -85,B 0,C 180,E1 -27210.563,E2 -27210.563} C_VEL
LIN {X 0,Y 139.203,Z 441.917,A -85,B 0,C 180,E1 -27211.501,E2 -27211.501} C_VEL
LIN {X 0,Y 135.707,Z 454.34,A -85,B 0,C 180,E1 -27212.732,E2 -27212.732} C_VEL
LIN {X 0,Y 131.833,Z 465.071,A -85,B 0,C 180,E1 -27214.285,E2 -27214.285} C_VEL
LIN {X 0,Y 126.602,Z 476.353,A -85,B 0,C 180,E1 -27216.402,E2 -27216.402} C_VEL
LIN {X 0,Y 120.961,Z 486.526,A -85,B 0,C 180,E1 -27219.009,E2 -27219.009} C_VEL
LIN {X 0,Y 115.572,Z 495.015,A -85,B 0,C 180,E1 -27221.984,E2 -27221.984} C_VEL
LIN {X 0,Y 109.031,Z 503.831,A -85,B 0,C 180,E1 -27226.143,E2 -27226.143} C_VEL
LIN {X 0,Y 102.801,Z 511.052,A -85,B 0,C 180,E1 -27230.78,E2 -27230.78} C_VEL
LIN {X 0,Y 96.581,Z 517.66,A -85,B 0,C 180,E1 -27236.929,E2 -27236.929} C_VEL
LIN {X 0,Y 92.102,Z 521.991,A -85,B 0,C 180,E1 -27242.757,E2 -27242.757} C_VEL
LIN {X 0,Y 89.671,Z 524.265,A -85,B 0,C 180,E1 -27246.934,E2 -27246.934} C_VEL
LIN {X 0,Y 87.691,Z 526.116,A -85,B 0,C 180,E1 -27251.307,E2 -27251.307} C_VEL
LIN {X 0,Y 86.17,Z 527.522,A -85,B 0,C 180,E1 -27255.842,E2 -27255.842} C_VEL
LIN {X 0,Y 84.473,Z 529.113,A -85,B 0,C 180,E1 -27265.232,E2 -27265.232} C_VEL
LIN {X 0,Y 84.299,Z 529.338,A -85,B 0,C 180,E1 -27270.005,E2 -27270.005} C_VEL
LIN {X 0,Y 84.474,Z 529.14,A -85,B 0,C 180,E1 -27274.777,E2 -27274.777} C_VEL
LIN {X 0,Y 86.112,Z 527.588,A -85,B 0,C 180,E1 -27284.177,E2 -27284.177} C_VEL
LIN {X 0,Y 87.632,Z 526.218,A -85,B 0,C 180,E1 -27288.716,E2 -27288.716} C_VEL
LIN {X 0,Y 90.795,Z 523.338,A -85,B 0,C 180,E1 -27295.202,E2 -27295.202} C_VEL
LIN {X 0,Y 94.949,Z 519.416,A -85,B 0,C 180,E1 -27301.212,E2 -27301.212} C_VEL
LIN {X 0,Y 99.94,Z 514.333,A -85,B 0,C 180,E1 -27306.713,E2 -27306.713} C_VEL
LIN {X 0,Y 105.782,Z 507.917,A -85,B 0,C 180,E1 -27311.64,E2 -27311.64} C_VEL
LIN {X 0,Y 112.105,Z 500.163,A -85,B 0,C 180,E1 -27315.924,E2 -27315.924} C_VEL
LIN {X 0,Y 117.909,Z 491.747,A -85,B 0,C 180,E1 -27319.465,E2 -27319.465} C_VEL
LIN {X 0,Y 124.042,Z 481.64,A -85,B 0,C 180,E1 -27322.492,E2 -27322.492} C_VEL
LIN {X 0,Y 129.807,Z 470.268,A -85,B 0,C 180,E1 -27324.979,E2 -27324.979} C_VEL
LIN {X 0,Y 134.384,Z 458.97,A -85,B 0,C 180,E1 -27326.805,E2 -27326.805} C_VEL
LIN {X 0,Y 135.78,Z 454.917,A -85,B 0,C 180,E1 -27327.339,E2 -27327.339} C_VEL
LIN {X 0,Y 135.823,Z 453.204,A -85,B 0,C 180,E1 -27327.882,E2 -27327.882} C_VEL
LIN {X 0,Y 131.002,Z 459.232,A -85,B 0,C 180,E1 -27329.139,E2 -27329.139} C_VEL
LIN {X 0,Y 125.645,Z 464.652,A -85,B 0,C 180,E1 -27330.961,E2 -27330.961} C_VEL
LIN {X 0,Y 119.62,Z 469.387,A -85,B 0,C 180,E1 -27333.855,E2 -27333.855} C_VEL
LIN {X 0,Y 114.109,Z 474.469,A -85,B 0,C 180,E1 -27336.208,E2 -27336.208} C_VEL
LIN {X 0,Y 111.323,Z 476.709,A -85,B 0,C 180,E1 -27337.741,E2 -27337.741} C_VEL
LIN {X 0,Y 107.379,Z 479.251,A -85,B 0,C 180,E1 -27340.898,E2 -27340.898} C_VEL
LIN {X 0,Y 105.341,Z 480.795,A -85,B 0,C 180,E1 -27342.529,E2 -27342.529} C_VEL
LIN {X 0,Y 103.048,Z 482.705,A -85,B 0,C 180,E1 -27344.168,E2 -27344.168} C_VEL
LIN {X 0,Y 99.946,Z 484.893,A -85,B 0,C 180,E1 -27347.822,E2 -27347.822} C_VEL
LIN {X 0,Y 98.767,Z 485.693,A -85,B 0,C 180,E1 -27349.753,E2 -27349.753} C_VEL
LIN {X 0,Y 97.166,Z 487.104,A -85,B 0,C 180,E1 -27351.682,E2 -27351.682} C_VEL
LIN {X 0,Y 95.015,Z 489.066,A -85,B 0,C 180,E1 -27355.758,E2 -27355.758} C_VEL
LIN {X 0,Y 93.722,Z 490.597,A -85,B 0,C 180,E1 -27360,E2 -27360} C_VEL
LIN {X 0,Y 92.64,Z 492.018,A -85,B 0,C 180,E1 -27362.174,E2 -27362.174} C_VEL
LIN {X 0,Y 91.898,Z 493.606,A -85,B 0,C 180,E1 -27366.143,E2 -27366.143} C_VEL
LIN {X 0,Y 92.027,Z 495.073,A -85,B 0,C 180,E1 -27371.006,E2 -27371.006} C_VEL
LIN {X 0,Y 91.476,Z 497.648,A -85,B 0,C 180,E1 -27375.599,E2 -27375.599} C_VEL
LIN {X 0,Y 91.762,Z 498.556,A -85,B 0,C 180,E1 -27377.84,E2 -27377.84} C_VEL
LIN {X 0,Y 93.743,Z 499.304,A -85,B 0,C 180,E1 -27382.015,E2 -27382.015} C_VEL
LIN {X 0,Y 94.277,Z 499.341,A -85,B 0,C 180,E1 -27382.605,E2 -27382.605} C_VEL
LIN {X 0,Y 99.209,Z 508.501,A -85,B 0,C 180,E1 -27390.823,E2 -27390.823} C_VEL
LIN {X 0,Y 106.988,Z 516.685,A -85,B 0,C 180,E1 -27398.612,E2 -27398.612} C_VEL
LIN {X 0,Y 113.425,Z 521.292,A -85,B 0,C 180,E1 -27402.967,E2 -27402.967} C_VEL
LIN {X 0,Y 113.851,Z 521.7,A -85,B 0,C 180,E1 -27404.232,E2 -27404.232} C_VEL
LIN {X 0,Y 105.457,Z 517.163,A -85,B 0,C 180,E1 -27410.561,E2 -27410.561} C_VEL
LIN {X 0,Y 100.585,Z 521.448,A -85,B 0,C 180,E1 -27413.561,E2 -27413.561} C_VEL
LIN {X 0,Y 94.665,Z 526.601,A -85,B 0,C 180,E1 -27418.684,E2 -27418.684} C_VEL
LIN {X 0,Y 90.139,Z 530.608,A -85,B 0,C 180,E1 -27424.602,E2 -27424.602} C_VEL
LIN {X 0,Y 86.856,Z 533.572,A -85,B 0,C 180,E1 -27431.111,E2 -27431.111} C_VEL
LIN {X 0,Y 85.362,Z 534.997,A -85,B 0,C 180,E1 -27435.696,E2 -27435.696} C_VEL
LIN {X 0,Y 84.089,Z 536.638,A -85,B 0,C 180,E1 -27445.201,E2 -27445.201} C_VEL
LIN {X 0,Y 84.188,Z 536.865,A -85,B 0,C 180,E1 -27449.995,E2 -27449.995} C_VEL
LIN {X 0,Y 83.967,Z 536.615,A -85,B 0,C 180,E1 -27454.796,E2 -27454.796} C_VEL
LIN {X 0,Y 84.818,Z 534.93,A -85,B 0,C 180,E1 -27464.388,E2 -27464.388} C_VEL
LIN {X 0,Y 86.015,Z 533.466,A -85,B 0,C 180,E1 -27469.071,E2 -27469.071} C_VEL
LIN {X 0,Y 88.869,Z 530.454,A -85,B 0,C 180,E1 -27475.777,E2 -27475.777} C_VEL
LIN {X 0,Y 92.85,Z 526.388,A -85,B 0,C 180,E1 -27481.99,E2 -27481.99} C_VEL
LIN {X 0,Y 98.245,Z 520.625,A -85,B 0,C 180,E1 -27488.104,E2 -27488.104} C_VEL
LIN {X 0,Y 104.591,Z 513.32,A -85,B 0,C 180,E1 -27493.526,E2 -27493.526} C_VEL
LIN {X 0,Y 111.289,Z 504.817,A -85,B 0,C 180,E1 -27497.898,E2 -27497.898} C_VEL
LIN {X 0,Y 117.353,Z 496.082,A -85,B 0,C 180,E1 -27501.121,E2 -27501.121} C_VEL
LIN {X 0,Y 123.825,Z 485.34,A -85,B 0,C 180,E1 -27503.973,E2 -27503.973} C_VEL
LIN {X 0,Y 129.202,Z 474.495,A -85,B 0,C 180,E1 -27506.044,E2 -27506.044} C_VEL
LIN {X 0,Y 134.048,Z 462.39,A -85,B 0,C 180,E1 -27507.71,E2 -27507.71} C_VEL
LIN {X 0,Y 137.579,Z 450.991,A -85,B 0,C 180,E1 -27508.825,E2 -27508.825} C_VEL
LIN {X 0,Y 140.41,Z 438.139,A -85,B 0,C 180,E1 -27509.654,E2 -27509.654} C_VEL
LIN {X 0,Y 142.278,Z 422.389,A -85,B 0,C 180,E1 -27510.333,E2 -27510.333} C_VEL
LIN {X 0,Y 142.997,Z 414.514,A -85,B 0,C 180,E1 -27510.609,E2 -27510.609} C_VEL
LIN {X 0,Y 142.918,Z 412.158,A -85,B 0,C 180,E1 -27510.901,E2 -27510.901} C_VEL
LIN {X 0,Y 142.036,Z 409.263,A -85,B 0,C 180,E1 -27511.84,E2 -27511.84} C_VEL
LIN {X 0,Y 140.715,Z 407.131,A -85,B 0,C 180,E1 -27513.084,E2 -27513.084} C_VEL
LIN {X 0,Y 137.234,Z 402.59,A -85,B 0,C 180,E1 -27516.647,E2 -27516.647} C_VEL
LIN {X 0,Y 136.859,Z 401.729,A -85,B 0,C 180,E1 -27517.122,E2 -27517.122} C_VEL
LIN {X 0,Y 134.07,Z 396.099,A -85,B 0,C 180,E1 -27520.975,E2 -27520.975} C_VEL
LIN {X 0,Y 131.747,Z 391.98,A -85,B 0,C 180,E1 -27524.927,E2 -27524.927} C_VEL
LIN {X 0,Y 130.143,Z 388.766,A -85,B 0,C 180,E1 -27528.596,E2 -27528.596} C_VEL
LIN {X 0,Y 128.556,Z 385.864,A -85,B 0,C 180,E1 -27534.117,E2 -27534.117} C_VEL
LIN {X 0,Y 128.307,Z 384.43,A -85,B 0,C 180,E1 -27536.271,E2 -27536.271} C_VEL
LIN {X 0,Y 128.054,Z 384.302,A -85,B 0,C 180,E1 -27541.573,E2 -27541.573} C_VEL
LIN {X 0,Y 128.354,Z 384.778,A -85,B 0,C 180,E1 -27544.711,E2 -27544.711} C_VEL
LIN {X 0,Y 129.37,Z 387.883,A -85,B 0,C 180,E1 -27549.774,E2 -27549.774} C_VEL
LIN {X 0,Y 130.369,Z 389.232,A -85,B 0,C 180,E1 -27552.453,E2 -27552.453} C_VEL
LIN {X 0,Y 132.7,Z 393.696,A -85,B 0,C 180,E1 -27557.283,E2 -27557.283} C_VEL
LIN {X 0,Y 134.663,Z 397.418,A -85,B 0,C 180,E1 -27560.396,E2 -27560.396} C_VEL
LIN {X 0,Y 137.548,Z 403.267,A -85,B 0,C 180,E1 -27564.197,E2 -27564.197} C_VEL
LIN {X 0,Y 140.286,Z 409.501,A -85,B 0,C 180,E1 -27567.295,E2 -27567.295} C_VEL
LIN {X 0,Y 138.185,Z 429.279,A -85,B 0,C 180,E1 -27568.075,E2 -27568.075} C_VEL
LIN {X 0,Y 135.511,Z 442.723,A -85,B 0,C 180,E1 -27568.99,E2 -27568.99} C_VEL
LIN {X 0,Y 131.939,Z 454.868,A -85,B 0,C 180,E1 -27570.174,E2 -27570.174} C_VEL
LIN {X 0,Y 127.982,Z 465.376,A -85,B 0,C 180,E1 -27571.668,E2 -27571.668} C_VEL
LIN {X 0,Y 122.532,Z 476.663,A -85,B 0,C 180,E1 -27573.736,E2 -27573.736} C_VEL
LIN {X 0,Y 116.624,Z 486.839,A -85,B 0,C 180,E1 -27576.299,E2 -27576.299} C_VEL
LIN {X 0,Y 110.568,Z 495.854,A -85,B 0,C 180,E1 -27579.467,E2 -27579.467} C_VEL
LIN {X 0,Y 104.033,Z 504.146,A -85,B 0,C 180,E1 -27583.435,E2 -27583.435} C_VEL
LIN {X 0,Y 97.421,Z 511.368,A -85,B 0,C 180,E1 -27588.147,E2 -27588.147} C_VEL
LIN {X 0,Y 90.699,Z 517.978,A -85,B 0,C 180,E1 -27594.474,E2 -27594.474} C_VEL
LIN {X 0,Y 85.865,Z 522.308,A -85,B 0,C 180,E1 -27600.593,E2 -27600.593} C_VEL
LIN {X 0,Y 83.202,Z 524.581,A -85,B 0,C 180,E1 -27605.023,E2 -27605.023} C_VEL
LIN {X 0,Y 80.992,Z 526.433,A -85,B 0,C 180,E1 -27609.696,E2 -27609.696} C_VEL
LIN {X 0,Y 79.305,Z 527.839,A -85,B 0,C 180,E1 -27614.587,E2 -27614.587} C_VEL
LIN {X 0,Y 77.424,Z 529.429,A -85,B 0,C 180,E1 -27624.797,E2 -27624.797} C_VEL
LIN {X 0,Y 77.225,Z 529.654,A -85,B 0,C 180,E1 -27630.005,E2 -27630.005} C_VEL
LIN {X 0,Y 77.425,Z 529.456,A -85,B 0,C 180,E1 -27635.213,E2 -27635.213} C_VEL
LIN {X 0,Y 79.261,Z 527.904,A -85,B 0,C 180,E1 -27645.432,E2 -27645.432} C_VEL
LIN {X 0,Y 80.945,Z 526.533,A -85,B 0,C 180,E1 -27650.327,E2 -27650.327} C_VEL
LIN {X 0,Y 84.427,Z 523.653,A -85,B 0,C 180,E1 -27657.253,E2 -27657.253} C_VEL
LIN {X 0,Y 88.948,Z 519.731,A -85,B 0,C 180,E1 -27663.584,E2 -27663.584} C_VEL
LIN {X 0,Y 94.357,Z 514.646,A -85,B 0,C 180,E1 -27669.285,E2 -27669.285} C_VEL
LIN {X 0,Y 100.602,Z 508.228,A -85,B 0,C 180,E1 -27674.319,E2 -27674.319} C_VEL
LIN {X 0,Y 107.089,Z 500.714,A -85,B 0,C 180,E1 -27678.534,E2 -27678.534} C_VEL
LIN {X 0,Y 113.419,Z 492.056,A -85,B 0,C 180,E1 -27682.195,E2 -27682.195} C_VEL
LIN {X 0,Y 119.85,Z 481.945,A -85,B 0,C 180,E1 -27685.186,E2 -27685.186} C_VEL
LIN {X 0,Y 125.994,Z 470.336,A -85,B 0,C 180,E1 -27687.661,E2 -27687.661} C_VEL
LIN {X 0,Y 126.375,Z 468.639,A -85,B 0,C 180,E1 -27688.262,E2 -27688.262} C_VEL
LIN {X 0,Y 118.163,Z 474.796,A -85,B 0,C 180,E1 -27691.587,E2 -27691.587} C_VEL
LIN {X 0,Y 112.085,Z 479.73,A -85,B 0,C 180,E1 -27693.965,E2 -27693.965} C_VEL
LIN {X 0,Y 109.363,Z 481.657,A -85,B 0,C 180,E1 -27695.31,E2 -27695.31} C_VEL
LIN {X 0,Y 102.821,Z 485.616,A -85,B 0,C 180,E1 -27700.016,E2 -27700.016} C_VEL
LIN {X 0,Y 100.335,Z 487.45,A -85,B 0,C 180,E1 -27701.627,E2 -27701.627} C_VEL
LIN {X 0,Y 98.399,Z 488.703,A -85,B 0,C 180,E1 -27703.399,E2 -27703.399} C_VEL
LIN {X 0,Y 95.333,Z 490.518,A -85,B 0,C 180,E1 -27707.222,E2 -27707.222} C_VEL
LIN {X 0,Y 92.296,Z 492.736,A -85,B 0,C 180,E1 -27711.24,E2 -27711.24} C_VEL
LIN {X 0,Y 87.011,Z 498.263,A -85,B 0,C 180,E1 -27724.633,E2 -27724.633} C_VEL
LIN {X 0,Y 86.862,Z 499.556,A -85,B 0,C 180,E1 -27729.312,E2 -27729.312} C_VEL
LIN {X 0,Y 86.165,Z 501.849,A -85,B 0,C 180,E1 -27734.164,E2 -27734.164} C_VEL
LIN {X 0,Y 86.824,Z 503.433,A -85,B 0,C 180,E1 -27738.892,E2 -27738.892} C_VEL
LIN {X 0,Y 88.753,Z 504.306,A -85,B 0,C 180,E1 -27743.324,E2 -27743.324} C_VEL
LIN {X 0,Y 89.917,Z 506.355,A -85,B 0,C 180,E1 -27747.967,E2 -27747.967} C_VEL
LIN {X 0,Y 92.429,Z 507.638,A -85,B 0,C 180,E1 -27752.158,E2 -27752.158} C_VEL
LIN {X 0,Y 95.904,Z 508.045,A -85,B 0,C 180,E1 -27755.358,E2 -27755.358} C_VEL
LIN {X 0,Y 104.045,Z 515.721,A -85,B 0,C 180,E1 -27762.491,E2 -27762.491} C_VEL
LIN {X 0,Y 105.831,Z 517.035,A -85,B 0,C 180,E1 -27763.673,E2 -27763.673} C_VEL
LIN {X 0,Y 104.355,Z 516.285,A -85,B 0,C 180,E1 -27765.222,E2 -27765.222} C_VEL
LIN {X 0,Y 102.034,Z 515.132,A -85,B 0,C 180,E1 -27766.969,E2 -27766.969} C_VEL
LIN {X 0,Y 94.988,Z 521.135,A -85,B 0,C 180,E1 -27771.026,E2 -27771.026} C_VEL
LIN {X 0,Y 88.682,Z 526.286,A -85,B 0,C 180,E1 -27776.301,E2 -27776.301} C_VEL
LIN {X 0,Y 83.79,Z 530.293,A -85,B 0,C 180,E1 -27782.522,E2 -27782.522} C_VEL
LIN {X 0,Y 80.164,Z 533.256,A -85,B 0,C 180,E1 -27789.466,E2 -27789.466} C_VEL
LIN {X 0,Y 78.497,Z 534.681,A -85,B 0,C 180,E1 -27794.414,E2 -27794.414} C_VEL
LIN {X 0,Y 77.01,Z 536.321,A -85,B 0,C 180,E1 -27804.759,E2 -27804.759} C_VEL
LIN {X 0,Y 77.076,Z 536.547,A -85,B 0,C 180,E1 -27809.995,E2 -27809.995} C_VEL
LIN {X 0,Y 76.879,Z 536.297,A -85,B 0,C 180,E1 -27815.24,E2 -27815.24} C_VEL
LIN {X 0,Y 77.926,Z 534.611,A -85,B 0,C 180,E1 -27825.692,E2 -27825.692} C_VEL
LIN {X 0,Y 79.285,Z 533.146,A -85,B 0,C 180,E1 -27830.761,E2 -27830.761} C_VEL
LIN {X 0,Y 82.515,Z 530.136,A -85,B 0,C 180,E1 -27837.928,E2 -27837.928} C_VEL
LIN {X 0,Y 86.891,Z 526.069,A -85,B 0,C 180,E1 -27844.479,E2 -27844.479} C_VEL
LIN {X 0,Y 92.273,Z 520.786,A -85,B 0,C 180,E1 -27850.39,E2 -27850.39} C_VEL
LIN {X 0,Y 99.547,Z 513.003,A -85,B 0,C 180,E1 -27856.35,E2 -27856.35} C_VEL
LIN {X 0,Y 106.637,Z 504.501,A -85,B 0,C 180,E1 -27860.744,E2 -27860.744} C_VEL
LIN {X 0,Y 113.021,Z 495.768,A -85,B 0,C 180,E1 -27863.931,E2 -27863.931} C_VEL
LIN {X 0,Y 119.789,Z 485.029,A -85,B 0,C 180,E1 -27866.718,E2 -27866.718} C_VEL
LIN {X 0,Y 125.38,Z 474.187,A -85,B 0,C 180,E1 -27868.733,E2 -27868.733} C_VEL
LIN {X 0,Y 130.369,Z 462.105,A -85,B 0,C 180,E1 -27870.36,E2 -27870.36} C_VEL
LIN {X 0,Y 134.268,Z 449.86,A -85,B 0,C 180,E1 -27871.489,E2 -27871.489} C_VEL
LIN {X 0,Y 137.09,Z 437.049,A -85,B 0,C 180,E1 -27872.265,E2 -27872.265} C_VEL
LIN {X 0,Y 139.009,Z 421.081,A -85,B 0,C 180,E1 -27872.911,E2 -27872.911} C_VEL
LIN {X 0,Y 140.081,Z 408.932,A -85,B 0,C 180,E1 -27873.393,E2 -27873.393} C_VEL
LIN {X 0,Y 136.859,Z 401.729,A -85,B 0,C 180,E1 -27877.122,E2 -27877.122} C_VEL
LIN {X 0,Y 135.832,Z 399.653,A -85,B 0,C 180,E1 -27878.448,E2 -27878.448} C_VEL
LIN {X 0,Y 134.097,Z 397.681,A -85,B 0,C 180,E1 -27880.693,E2 -27880.693} C_VEL
LIN {X 0,Y 132.363,Z 396.7,A -85,B 0,C 180,E1 -27883.107,E2 -27883.107} C_VEL
LIN {X 0,Y 128.672,Z 395.261,A -85,B 0,C 180,E1 -27890.114,E2 -27890.114} C_VEL
LIN {X 0,Y 127.451,Z 392.08,A -85,B 0,C 180,E1 -27895.751,E2 -27895.751} C_VEL
LIN {X 0,Y 127.362,Z 391.451,A -85,B 0,C 180,E1 -27896.837,E2 -27896.837} C_VEL
LIN {X 0,Y 127.189,Z 391.352,A -85,B 0,C 180,E1 -27901.583,E2 -27901.583} C_VEL
LIN {X 0,Y 127.398,Z 391.795,A -85,B 0,C 180,E1 -27904.152,E2 -27904.152} C_VEL
LIN {X 0,Y 128.5,Z 395.074,A -85,B 0,C 180,E1 -27909.841,E2 -27909.841} C_VEL
LIN {X 0,Y 129.139,Z 396.046,A -85,B 0,C 180,E1 -27911.663,E2 -27911.663} C_VEL
LIN {X 0,Y 131.103,Z 400.114,A -85,B 0,C 180,E1 -27916.146,E2 -27916.146} C_VEL
LIN {X 0,Y 133.451,Z 404.878,A -85,B 0,C 180,E1 -27920.118,E2 -27920.118} C_VEL
LIN {X 0,Y 135.953,Z 410.643,A -85,B 0,C 180,E1 -27923.618,E2 -27923.618} C_VEL
LIN {X 0,Y 136.861,Z 412.849,A -85,B 0,C 180,E1 -27924.757,E2 -27924.757} C_VEL
LIN {X 0,Y 134.988,Z 429.551,A -85,B 0,C 180,E1 -27925.414,E2 -27925.414} C_VEL
LIN {X 0,Y 132.224,Z 443.013,A -85,B 0,C 180,E1 -27926.305,E2 -27926.305} C_VEL
LIN {X 0,Y 128.445,Z 455.396,A -85,B 0,C 180,E1 -27927.47,E2 -27927.47} C_VEL
LIN {X 0,Y 123.696,Z 467.218,A -85,B 0,C 180,E1 -27929.132,E2 -27929.132} C_VEL
LIN {X 0,Y 118.052,Z 478.229,A -85,B 0,C 180,E1 -27931.16,E2 -27931.16} C_VEL
LIN {X 0,Y 111.915,Z 488.171,A -85,B 0,C 180,E1 -27933.696,E2 -27933.696} C_VEL
LIN {X 0,Y 105.467,Z 497.099,A -85,B 0,C 180,E1 -27936.911,E2 -27936.911} C_VEL
LIN {X 0,Y 98.093,Z 505.785,A -85,B 0,C 180,E1 -27941.218,E2 -27941.218} C_VEL
LIN {X 0,Y 91.153,Z 512.762,A -85,B 0,C 180,E1 -27946.066,E2 -27946.066} C_VEL
LIN {X 0,Y 85.013,Z 518.295,A -85,B 0,C 180,E1 -27951.689,E2 -27951.689} C_VEL
LIN {X 0,Y 79.772,Z 522.624,A -85,B 0,C 180,E1 -27958.095,E2 -27958.095} C_VEL
LIN {X 0,Y 76.817,Z 524.899,A -85,B 0,C 180,E1 -27962.783,E2 -27962.783} C_VEL
LIN {X 0,Y 74.382,Z 526.751,A -85,B 0,C 180,E1 -27967.8,E2 -27967.8} C_VEL
LIN {X 0,Y 72.5,Z 528.156,A -85,B 0,C 180,E1 -27973.099,E2 -27973.099} C_VEL
LIN {X 0,Y 70.378,Z 529.746,A -85,B 0,C 180,E1 -27984.275,E2 -27984.275} C_VEL
LIN {X 0,Y 70.137,Z 529.971,A -85,B 0,C 180,E1 -27990.006,E2 -27990.006} C_VEL
LIN {X 0,Y 70.379,Z 529.772,A -85,B 0,C 180,E1 -27995.737,E2 -27995.737} C_VEL
LIN {X 0,Y 72.45,Z 528.22,A -85,B 0,C 180,E1 -28006.925,E2 -28006.925} C_VEL
LIN {X 0,Y 74.342,Z 526.849,A -85,B 0,C 180,E1 -28012.224,E2 -28012.224} C_VEL
LIN {X 0,Y 78.175,Z 523.969,A -85,B 0,C 180,E1 -28019.639,E2 -28019.639} C_VEL
LIN {X 0,Y 83.125,Z 520.045,A -85,B 0,C 180,E1 -28026.293,E2 -28026.293} C_VEL
LIN {X 0,Y 88.968,Z 514.96,A -85,B 0,C 180,E1 -28032.185,E2 -28032.185} C_VEL
LIN {X 0,Y 95.668,Z 508.539,A -85,B 0,C 180,E1 -28037.281,E2 -28037.281} C_VEL
LIN {X 0,Y 102.329,Z 501.265,A -85,B 0,C 180,E1 -28041.386,E2 -28041.386} C_VEL
LIN {X 0,Y 109.224,Z 492.361,A -85,B 0,C 180,E1 -28045.13,E2 -28045.13} C_VEL
LIN {X 0,Y 115.957,Z 482.248,A -85,B 0,C 180,E1 -28048.057,E2 -28048.057} C_VEL
LIN {X 0,Y 116.72,Z 480.964,A -85,B 0,C 180,E1 -28048.373,E2 -28048.373} C_VEL
LIN {X 0,Y 116.985,Z 479.722,A -85,B 0,C 180,E1 -28049.092,E2 -28049.092} C_VEL
LIN {X 0,Y 110.28,Z 484.578,A -85,B 0,C 180,E1 -28051.445,E2 -28051.445} C_VEL
LIN {X 0,Y 107.388,Z 486.411,A -85,B 0,C 180,E1 -28052.734,E2 -28052.734} C_VEL
LIN {X 0,Y 100.025,Z 490.397,A -85,B 0,C 180,E1 -28057.484,E2 -28057.484} C_VEL
LIN {X 0,Y 97.602,Z 492.001,A -85,B 0,C 180,E1 -28058.897,E2 -28058.897} C_VEL
LIN {X 0,Y 93.599,Z 494.188,A -85,B 0,C 180,E1 -28062.521,E2 -28062.521} C_VEL
LIN {X 0,Y 82.844,Z 501.57,A -85,B 0,C 180,E1 -28080,E2 -28080} C_VEL
LIN {X 0,Y 81.15,Z 504.702,A -85,B 0,C 180,E1 -28089.974,E2 -28089.974} C_VEL
LIN {X 0,Y 80.969,Z 507.297,A -85,B 0,C 180,E1 -28097.28,E2 -28097.28} C_VEL
LIN {X 0,Y 83.237,Z 509.201,A -85,B 0,C 180,E1 -28104.972,E2 -28104.972} C_VEL
LIN {X 0,Y 84.885,Z 510.867,A -85,B 0,C 180,E1 -28109.786,E2 -28109.786} C_VEL
LIN {X 0,Y 87.698,Z 511.957,A -85,B 0,C 180,E1 -28114.123,E2 -28114.123} C_VEL
LIN {X 0,Y 91.261,Z 512.761,A -85,B 0,C 180,E1 -28118.03,E2 -28118.03} C_VEL
LIN {X 0,Y 95.608,Z 514.377,A -85,B 0,C 180,E1 -28122.837,E2 -28122.837} C_VEL
LIN {X 0,Y 95.959,Z 515.622,A -85,B 0,C 180,E1 -28124.502,E2 -28124.502} C_VEL
LIN {X 0,Y 89.602,Z 520.823,A -85,B 0,C 180,E1 -28128.181,E2 -28128.181} C_VEL
LIN {X 0,Y 82.873,Z 525.972,A -85,B 0,C 180,E1 -28133.579,E2 -28133.579} C_VEL
LIN {X 0,Y 77.571,Z 529.978,A -85,B 0,C 180,E1 -28140.107,E2 -28140.107} C_VEL
LIN {X 0,Y 73.559,Z 532.94,A -85,B 0,C 180,E1 -28147.526,E2 -28147.526} C_VEL
LIN {X 0,Y 71.688,Z 534.364,A -85,B 0,C 180,E1 -28152.89,E2 -28152.89} C_VEL
LIN {X 0,Y 69.932,Z 536.004,A -85,B 0,C 180,E1 -28164.226,E2 -28164.226} C_VEL
LIN {X 0,Y 69.967,Z 536.23,A -85,B 0,C 180,E1 -28169.994,E2 -28169.994} C_VEL
LIN {X 0,Y 69.787,Z 535.978,A -85,B 0,C 180,E1 -28175.774,E2 -28175.774} C_VEL
LIN {X 0,Y 71.09,Z 534.292,A -85,B 0,C 180,E1 -28187.246,E2 -28187.246} C_VEL
LIN {X 0,Y 72.641,Z 532.826,A -85,B 0,C 180,E1 -28192.762,E2 -28192.762} C_VEL
LIN {X 0,Y 76.274,Z 529.817,A -85,B 0,C 180,E1 -28200.443,E2 -28200.443} C_VEL
LIN {X 0,Y 81.121,Z 525.751,A -85,B 0,C 180,E1 -28207.327,E2 -28207.327} C_VEL
LIN {X 0,Y 87.161,Z 520.277,A -85,B 0,C 180,E1 -28213.613,E2 -28213.613} C_VEL
LIN {X 0,Y 94.762,Z 512.686,A -85,B 0,C 180,E1 -28219.474,E2 -28219.474} C_VEL
LIN {X 0,Y 102.279,Z 504.185,A -85,B 0,C 180,E1 -28223.834,E2 -28223.834} C_VEL
LIN {X 0,Y 108.986,Z 495.454,A -85,B 0,C 180,E1 -28226.955,E2 -28226.955} C_VEL
LIN {X 0,Y 116.046,Z 484.718,A -85,B 0,C 180,E1 -28229.649,E2 -28229.649} C_VEL
LIN {X 0,Y 121.845,Z 473.88,A -85,B 0,C 180,E1 -28231.588,E2 -28231.588} C_VEL
LIN {X 0,Y 126.962,Z 461.926,A -85,B 0,C 180,E1 -28233.13,E2 -28233.13} C_VEL
LIN {X 0,Y 130.967,Z 449.799,A -85,B 0,C 180,E1 -28234.2,E2 -28234.2} C_VEL
LIN {X 0,Y 133.808,Z 437.483,A -85,B 0,C 180,E1 -28234.923,E2 -28234.923} C_VEL
LIN {X 0,Y 135.724,Z 422.873,A -85,B 0,C 180,E1 -28235.507,E2 -28235.507} C_VEL
LIN {X 0,Y 136.698,Z 412.368,A -85,B 0,C 180,E1 -28235.915,E2 -28235.915} C_VEL
LIN {X 0,Y 133.821,Z 405.659,A -85,B 0,C 180,E1 -28239.791,E2 -28239.791} C_VEL
LIN {X 0,Y 131.739,Z 401.389,A -85,B 0,C 180,E1 -28243.137,E2 -28243.137} C_VEL
LIN {X 0,Y 130.226,Z 398.391,A -85,B 0,C 180,E1 -28246.104,E2 -28246.104} C_VEL
LIN {X 0,Y 128.835,Z 395.483,A -85,B 0,C 180,E1 -28249.652,E2 -28249.652} C_VEL
LIN {X 0,Y 128.672,Z 395.261,A -85,B 0,C 180,E1 -28250.114,E2 -28250.114} C_VEL
LIN {X 0,Y 127.582,Z 394.723,A -85,B 0,C 180,E1 -28253.637,E2 -28253.637} C_VEL
LIN {X 0,Y 126.822,Z 395.486,A -85,B 0,C 180,E1 -28257.206,E2 -28257.206} C_VEL
LIN {X 0,Y 126.422,Z 398.16,A -85,B 0,C 180,E1 -28262.555,E2 -28262.555} C_VEL
LIN {X 0,Y 126.505,Z 399.258,A -85,B 0,C 180,E1 -28264.318,E2 -28264.318} C_VEL
LIN {X 0,Y 127.998,Z 403.039,A -85,B 0,C 180,E1 -28271.06,E2 -28271.06} C_VEL
LIN {X 0,Y 129.674,Z 406.755,A -85,B 0,C 180,E1 -28275.22,E2 -28275.22} C_VEL
LIN {X 0,Y 131.636,Z 411.158,A -85,B 0,C 180,E1 -28278.885,E2 -28278.885} C_VEL
LIN {X 0,Y 133.693,Z 416.328,A -85,B 0,C 180,E1 -28282.085,E2 -28282.085} C_VEL
LIN {X 0,Y 131.858,Z 431.194,A -85,B 0,C 180,E1 -28282.705,E2 -28282.705} C_VEL
LIN {X 0,Y 128.898,Z 444.644,A -85,B 0,C 180,E1 -28283.592,E2 -28283.592} C_VEL
LIN {X 0,Y 125.251,Z 455.927,A -85,B 0,C 180,E1 -28284.624,E2 -28284.624} C_VEL
LIN {X 0,Y 120.411,Z 467.525,A -85,B 0,C 180,E1 -28286.191,E2 -28286.191} C_VEL
LIN {X 0,Y 114.554,Z 478.539,A -85,B 0,C 180,E1 -28288.133,E2 -28288.133} C_VEL
LIN {X 0,Y 108.137,Z 488.485,A -85,B 0,C 180,E1 -28290.563,E2 -28290.563} C_VEL
LIN {X 0,Y 101.353,Z 497.415,A -85,B 0,C 180,E1 -28293.693,E2 -28293.693} C_VEL
LIN {X 0,Y 93.576,Z 506.1,A -85,B 0,C 180,E1 -28297.953,E2 -28297.953} C_VEL
LIN {X 0,Y 86.197,Z 513.078,A -85,B 0,C 180,E1 -28302.801,E2 -28302.801} C_VEL
LIN {X 0,Y 79.562,Z 518.612,A -85,B 0,C 180,E1 -28308.516,E2 -28308.516} C_VEL
LIN {X 0,Y 73.843,Z 522.941,A -85,B 0,C 180,E1 -28315.183,E2 -28315.183} C_VEL
LIN {X 0,Y 70.579,Z 525.216,A -85,B 0,C 180,E1 -28320.147,E2 -28320.147} C_VEL
LIN {X 0,Y 67.877,Z 527.067,A -85,B 0,C 180,E1 -28325.54,E2 -28325.54} C_VEL
LIN {X 0,Y 65.748,Z 528.473,A -85,B 0,C 180,E1 -28331.303,E2 -28331.303} C_VEL
LIN {X 0,Y 63.326,Z 530.062,A -85,B 0,C 180,E1 -28343.635,E2 -28343.635} C_VEL
LIN {X 0,Y 63.057,Z 530.287,A -85,B 0,C 180,E1 -28350.006,E2 -28350.006} C_VEL
LIN {X 0,Y 63.327,Z 530.088,A -85,B 0,C 180,E1 -28356.378,E2 -28356.378} C_VEL
LIN {X 0,Y 65.685,Z 528.537,A -85,B 0,C 180,E1 -28368.729,E2 -28368.729} C_VEL
LIN {X 0,Y 67.819,Z 527.165,A -85,B 0,C 180,E1 -28374.495,E2 -28374.495} C_VEL
LIN {X 0,Y 72.084,Z 524.285,A -85,B 0,C 180,E1 -28382.434,E2 -28382.434} C_VEL
LIN {X 0,Y 77.52,Z 520.36,A -85,B 0,C 180,E1 -28389.398,E2 -28389.398} C_VEL
LIN {X 0,Y 83.84,Z 515.274,A -85,B 0,C 180,E1 -28395.447,E2 -28395.447} C_VEL
LIN {X 0,Y 91.006,Z 508.851,A -85,B 0,C 180,E1 -28400.564,E2 -28400.564} C_VEL
LIN {X 0,Y 97.619,Z 502.067,A -85,B 0,C 180,E1 -28404.389,E2 -28404.389} C_VEL
LIN {X 0,Y 105.327,Z 492.668,A -85,B 0,C 180,E1 -28408.302,E2 -28408.302} C_VEL
LIN {X 0,Y 106.698,Z 490.794,A -85,B 0,C 180,E1 -28408.909,E2 -28408.909} C_VEL
LIN {X 0,Y 105.574,Z 490.889,A -85,B 0,C 180,E1 -28409.935,E2 -28409.935} C_VEL
LIN {X 0,Y 97.739,Z 494.678,A -85,B 0,C 180,E1 -28414.441,E2 -28414.441} C_VEL
LIN {X 0,Y 94.494,Z 496.544,A -85,B 0,C 180,E1 -28416.238,E2 -28416.238} C_VEL
LIN {X 0,Y 84.834,Z 501.263,A -85,B 0,C 180,E1 -28425.609,E2 -28425.609} C_VEL
LIN {X 0,Y 75.262,Z 509.43,A -85,B 0,C 180,E1 -28450.764,E2 -28450.764} C_VEL
LIN {X 0,Y 75.049,Z 511.118,A -85,B 0,C 180,E1 -28456.316,E2 -28456.316} C_VEL
LIN {X 0,Y 77.752,Z 513.582,A -85,B 0,C 180,E1 -28466.869,E2 -28466.869} C_VEL
LIN {X 0,Y 79.764,Z 514.983,A -85,B 0,C 180,E1 -28471.915,E2 -28471.915} C_VEL
LIN {X 0,Y 87.367,Z 517.171,A -85,B 0,C 180,E1 -28481.598,E2 -28481.598} C_VEL
LIN {X 0,Y 87.629,Z 518.087,A -85,B 0,C 180,E1 -28483.083,E2 -28483.083} C_VEL
LIN {X 0,Y 79.569,Z 524.063,A -85,B 0,C 180,E1 -28488.507,E2 -28488.507} C_VEL
LIN {X 0,Y 73.279,Z 528.427,A -85,B 0,C 180,E1 -28494.863,E2 -28494.863} C_VEL
LIN {X 0,Y 69.861,Z 530.738,A -85,B 0,C 180,E1 -28499.795,E2 -28499.795} C_VEL
LIN {X 0,Y 67.061,Z 532.624,A -85,B 0,C 180,E1 -28505.209,E2 -28505.209} C_VEL
LIN {X 0,Y 64.92,Z 534.047,A -85,B 0,C 180,E1 -28511.042,E2 -28511.042} C_VEL
LIN {X 0,Y 62.882,Z 535.687,A -85,B 0,C 180,E1 -28523.577,E2 -28523.577} C_VEL
LIN {X 0,Y 62.858,Z 535.912,A -85,B 0,C 180,E1 -28529.994,E2 -28529.994} C_VEL
LIN {X 0,Y 62.704,Z 535.66,A -85,B 0,C 180,E1 -28536.429,E2 -28536.429} C_VEL
LIN {X 0,Y 64.29,Z 533.972,A -85,B 0,C 180,E1 -28549.138,E2 -28549.138} C_VEL
LIN {X 0,Y 66.107,Z 532.506,A -85,B 0,C 180,E1 -28555.159,E2 -28555.159} C_VEL
LIN {X 0,Y 70.211,Z 529.497,A -85,B 0,C 180,E1 -28563.397,E2 -28563.397} C_VEL
LIN {X 0,Y 75.577,Z 525.433,A -85,B 0,C 180,E1 -28570.605,E2 -28570.605} C_VEL
LIN {X 0,Y 82.914,Z 519.277,A -85,B 0,C 180,E1 -28577.686,E2 -28577.686} C_VEL
LIN {X 0,Y 90.294,Z 512.369,A -85,B 0,C 180,E1 -28582.913,E2 -28582.913} C_VEL
LIN {X 0,Y 98.251,Z 503.87,A -85,B 0,C 180,E1 -28587.184,E2 -28587.184} C_VEL
LIN {X 0,Y 105.281,Z 495.141,A -85,B 0,C 180,E1 -28590.197,E2 -28590.197} C_VEL
LIN {X 0,Y 112.621,Z 484.406,A -85,B 0,C 180,E1 -28592.771,E2 -28592.771} C_VEL
LIN {X 0,Y 118.63,Z 473.572,A -85,B 0,C 180,E1 -28594.607,E2 -28594.607} C_VEL
LIN {X 0,Y 123.869,Z 461.75,A -85,B 0,C 180,E1 -28596.042,E2 -28596.042} C_VEL
LIN {X 0,Y 128.137,Z 449.184,A -85,B 0,C 180,E1 -28597.072,E2 -28597.072} C_VEL
LIN {X 0,Y 131.156,Z 436.006,A -85,B 0,C 180,E1 -28597.81,E2 -28597.81} C_VEL
LIN {X 0,Y 133.252,Z 419.443,A -85,B 0,C 180,E1 -28598.41,E2 -28598.41} C_VEL
LIN {X 0,Y 133.556,Z 415.892,A -85,B 0,C 180,E1 -28598.588,E2 -28598.588} C_VEL
LIN {X 0,Y 131.343,Z 410.45,A -85,B 0,C 180,E1 -28602.081,E2 -28602.081} C_VEL
LIN {X 0,Y 129.612,Z 406.606,A -85,B 0,C 180,E1 -28605.376,E2 -28605.376} C_VEL
LIN {X 0,Y 127.654,Z 402.24,A -85,B 0,C 180,E1 -28610.493,E2 -28610.493} C_VEL
LIN {X 0,Y 126.509,Z 399.113,A -85,B 0,C 180,E1 -28616.218,E2 -28616.218} C_VEL
LIN {X 0,Y 126.414,Z 398.437,A -85,B 0,C 180,E1 -28617.61,E2 -28617.61} C_VEL
LIN {X 0,Y 126.323,Z 398.402,A -85,B 0,C 180,E1 -28621.594,E2 -28621.594} C_VEL
LIN {X 0,Y 126.459,Z 398.778,A -85,B 0,C 180,E1 -28623.585,E2 -28623.585} C_VEL
LIN {X 0,Y 126.505,Z 399.258,A -85,B 0,C 180,E1 -28624.318,E2 -28624.318} C_VEL
LIN {X 0,Y 126.753,Z 401.418,A -85,B 0,C 180,E1 -28626.814,E2 -28626.814} C_VEL
LIN {X 0,Y 127.372,Z 406.587,A -85,B 0,C 180,E1 -28630.624,E2 -28630.624} C_VEL
LIN {X 0,Y 129.27,Z 415.882,A -85,B 0,C 180,E1 -28636.426,E2 -28636.426} C_VEL
LIN {X 0,Y 130.836,Z 419.985,A -85,B 0,C 180,E1 -28639.327,E2 -28639.327} C_VEL
LIN {X 0,Y 128.842,Z 433.939,A -85,B 0,C 180,E1 -28639.932,E2 -28639.932} C_VEL
LIN {X 0,Y 125.855,Z 446.23,A -85,B 0,C 180,E1 -28640.746,E2 -28640.746} C_VEL
LIN {X 0,Y 121.827,Z 457.897,A -85,B 0,C 180,E1 -28641.823,E2 -28641.823} C_VEL
LIN {X 0,Y 116.698,Z 469.367,A -85,B 0,C 180,E1 -28643.314,E2 -28643.314} C_VEL
LIN {X 0,Y 110.625,Z 480.088,A -85,B 0,C 180,E1 -28645.145,E2 -28645.145} C_VEL
LIN {X 0,Y 103.259,Z 490.706,A -85,B 0,C 180,E1 -28647.782,E2 -28647.782} C_VEL
LIN {X 0,Y 95.504,Z 500.118,A -85,B 0,C 180,E1 -28651.206,E2 -28651.206} C_VEL
LIN {X 0,Y 88.052,Z 507.692,A -85,B 0,C 180,E1 -28655.112,E2 -28655.112} C_VEL
LIN {X 0,Y 81.555,Z 513.393,A -85,B 0,C 180,E1 -28659.151,E2 -28659.151} C_VEL
LIN {X 0,Y 74.394,Z 518.929,A -85,B 0,C 180,E1 -28664.893,E2 -28664.893} C_VEL
LIN {X 0,Y 68.127,Z 523.259,A -85,B 0,C 180,E1 -28671.768,E2 -28671.768} C_VEL
LIN {X 0,Y 64.524,Z 525.533,A -85,B 0,C 180,E1 -28677.01,E2 -28677.01} C_VEL
LIN {X 0,Y 61.481,Z 527.385,A -85,B 0,C 180,E1 -28682.798,E2 -28682.798} C_VEL
LIN {X 0,Y 59.062,Z 528.79,A -85,B 0,C 180,E1 -28689.093,E2 -28689.093} C_VEL
LIN {X 0,Y 56.294,Z 530.379,A -85,B 0,C 180,E1 -28702.836,E2 -28702.836} C_VEL
LIN {X 0,Y 55.977,Z 530.603,A -85,B 0,C 180,E1 -28710.007,E2 -28710.007} C_VEL
LIN {X 0,Y 56.294,Z 530.404,A -85,B 0,C 180,E1 -28717.179,E2 -28717.179} C_VEL
LIN {X 0,Y 59.008,Z 528.853,A -85,B 0,C 180,E1 -28730.942,E2 -28730.942} C_VEL
LIN {X 0,Y 61.434,Z 527.481,A -85,B 0,C 180,E1 -28737.239,E2 -28737.239} C_VEL
LIN {X 0,Y 66.198,Z 524.601,A -85,B 0,C 180,E1 -28745.734,E2 -28745.734} C_VEL
LIN {X 0,Y 72.164,Z 520.675,A -85,B 0,C 180,E1 -28752.986,E2 -28752.986} C_VEL
LIN {X 0,Y 79.023,Z 515.588,A -85,B 0,C 180,E1 -28759.117,E2 -28759.117} C_VEL
LIN {X 0,Y 86.67,Z 509.164,A -85,B 0,C 180,E1 -28764.191,E2 -28764.191} C_VEL
LIN {X 0,Y 94.774,Z 501.165,A -85,B 0,C 180,E1 -28768.527,E2 -28768.527} C_VEL
LIN {X 0,Y 97.549,Z 498.064,A -85,B 0,C 180,E1 -28769.839,E2 -28769.839} C_VEL
LIN {X 0,Y 97.003,Z 498.112,A -85,B 0,C 180,E1 -28770.399,E2 -28770.399} C_VEL
LIN {X 0,Y 89.674,Z 501.568,A -85,B 0,C 180,E1 -28774.465,E2 -28774.465} C_VEL
LIN {X 0,Y 75.95,Z 507.664,A -85,B 0,C 180,E1 -28789.335,E2 -28789.335} C_VEL
LIN {X 0,Y 69.239,Z 515.156,A -85,B 0,C 180,E1 -28817.729,E2 -28817.729} C_VEL
LIN {X 0,Y 72.208,Z 517.534,A -85,B 0,C 180,E1 -28829.121,E2 -28829.121} C_VEL
LIN {X 0,Y 74.592,Z 518.724,A -85,B 0,C 180,E1 -28834.424,E2 -28834.424} C_VEL
LIN {X 0,Y 77.949,Z 519.638,A -85,B 0,C 180,E1 -28839.133,E2 -28839.133} C_VEL
LIN {X 0,Y 79.233,Z 520.466,A -85,B 0,C 180,E1 -28841.582,E2 -28841.582} C_VEL
LIN {X 0,Y 71.953,Z 525.343,A -85,B 0,C 180,E1 -28846.857,E2 -28846.857} C_VEL
LIN {X 0,Y 65.649,Z 529.347,A -85,B 0,C 180,E1 -28853.921,E2 -28853.921} C_VEL
LIN {X 0,Y 60.687,Z 532.308,A -85,B 0,C 180,E1 -28862.397,E2 -28862.397} C_VEL
LIN {X 0,Y 58.243,Z 533.73,A -85,B 0,C 180,E1 -28868.77,E2 -28868.77} C_VEL
LIN {X 0,Y 55.826,Z 535.37,A -85,B 0,C 180,E1 -28882.761,E2 -28882.761} C_VEL
LIN {X 0,Y 55.758,Z 535.595,A -85,B 0,C 180,E1 -28889.993,E2 -28889.993} C_VEL
LIN {X 0,Y 55.618,Z 535.341,A -85,B 0,C 180,E1 -28897.252,E2 -28897.252} C_VEL
LIN {X 0,Y 57.581,Z 533.652,A -85,B 0,C 180,E1 -28911.472,E2 -28911.472} C_VEL
LIN {X 0,Y 59.718,Z 532.186,A -85,B 0,C 180,E1 -28918.075,E2 -28918.075} C_VEL
LIN {X 0,Y 64.371,Z 529.178,A -85,B 0,C 180,E1 -28926.897,E2 -28926.897} C_VEL
LIN {X 0,Y 70.318,Z 525.114,A -85,B 0,C 180,E1 -28934.388,E2 -28934.388} C_VEL
LIN {X 0,Y 78.283,Z 518.958,A -85,B 0,C 180,E1 -28941.555,E2 -28941.555} C_VEL
LIN {X 0,Y 86.178,Z 512.051,A -85,B 0,C 180,E1 -28946.702,E2 -28946.702} C_VEL
LIN {X 0,Y 94.585,Z 503.554,A -85,B 0,C 180,E1 -28950.808,E2 -28950.808} C_VEL
LIN {X 0,Y 101.939,Z 494.827,A -85,B 0,C 180,E1 -28953.661,E2 -28953.661} C_VEL
LIN {X 0,Y 109.551,Z 484.095,A -85,B 0,C 180,E1 -28956.079,E2 -28956.079} C_VEL
LIN {X 0,Y 115.763,Z 473.265,A -85,B 0,C 180,E1 -28957.783,E2 -28957.783} C_VEL
LIN {X 0,Y 121.11,Z 461.581,A -85,B 0,C 180,E1 -28959.094,E2 -28959.094} C_VEL
LIN {X 0,Y 125.539,Z 448.892,A -85,B 0,C 180,E1 -28960.06,E2 -28960.06} C_VEL
LIN {X 0,Y 128.612,Z 435.921,A -85,B 0,C 180,E1 -28960.726,E2 -28960.726} C_VEL
LIN {X 0,Y 130.639,Z 420.847,A -85,B 0,C 180,E1 -28961.245,E2 -28961.245} C_VEL
LIN {X 0,Y 130.698,Z 419.573,A -85,B 0,C 180,E1 -28961.381,E2 -28961.381} C_VEL
LIN {X 0,Y 128.828,Z 414.651,A -85,B 0,C 180,E1 -28964.982,E2 -28964.982} C_VEL
LIN {X 0,Y 127.309,Z 411.156,A -85,B 0,C 180,E1 -28968.658,E2 -28968.658} C_VEL
LIN {X 0,Y 126.539,Z 409.082,A -85,B 0,C 180,E1 -28971.215,E2 -28971.215} C_VEL
LIN {X 0,Y 125.546,Z 405.687,A -85,B 0,C 180,E1 -28977.393,E2 -28977.393} C_VEL
LIN {X 0,Y 125.437,Z 405.333,A -85,B 0,C 180,E1 -28980,E2 -28980} C_VEL
LIN {X 0,Y 125.534,Z 405.745,A -85,B 0,C 180,E1 -28983.009,E2 -28983.009} C_VEL
LIN {X 0,Y 126.518,Z 409.093,A -85,B 0,C 180,E1 -28989.19,E2 -28989.19} C_VEL
LIN {X 0,Y 128.154,Z 413.122,A -85,B 0,C 180,E1 -28993.984,E2 -28993.984} C_VEL
LIN {X 0,Y 129.27,Z 415.882,A -85,B 0,C 180,E1 -28996.426,E2 -28996.426} C_VEL
LIN {X 0,Y 129.524,Z 417.742,A -85,B 0,C 180,E1 -28997.155,E2 -28997.155} C_VEL
LIN {X 0,Y 129.421,Z 420.842,A -85,B 0,C 180,E1 -28997.584,E2 -28997.584} C_VEL
LIN {X 0,Y 128.727,Z 425.585,A -85,B 0,C 180,E1 -28997.579,E2 -28997.579} C_VEL
LIN {X 0,Y 126.528,Z 434.787,A -85,B 0,C 180,E1 -28996.995,E2 -28996.995} C_VEL
LIN {X 0,Y 126.021,Z 436.887,A -85,B 0,C 180,E1 -28997.048,E2 -28997.048} C_VEL
LIN {X 0,Y 122.68,Z 449.193,A -85,B 0,C 180,E1 -28997.884,E2 -28997.884} C_VEL
LIN {X 0,Y 118.79,Z 459.634,A -85,B 0,C 180,E1 -28998.818,E2 -28998.818} C_VEL
LIN {X 0,Y 113.291,Z 471.185,A -85,B 0,C 180,E1 -29000.247,E2 -29000.247} C_VEL
LIN {X 0,Y 106.25,Z 482.695,A -85,B 0,C 180,E1 -29002.185,E2 -29002.185} C_VEL
LIN {X 0,Y 98.649,Z 492.919,A -85,B 0,C 180,E1 -29004.734,E2 -29004.734} C_VEL
LIN {X 0,Y 89.97,Z 502.51,A -85,B 0,C 180,E1 -29008.328,E2 -29008.328} C_VEL
LIN {X 0,Y 81.363,Z 510.42,A -85,B 0,C 180,E1 -29012.638,E2 -29012.638} C_VEL
LIN {X 0,Y 74.608,Z 515.69,A -85,B 0,C 180,E1 -29016.814,E2 -29016.814} C_VEL
LIN {X 0,Y 67.187,Z 520.825,A -85,B 0,C 180,E1 -29022.936,E2 -29022.936} C_VEL
LIN {X 0,Y 60.624,Z 524.788,A -85,B 0,C 180,E1 -29030.395,E2 -29030.395} C_VEL
LIN {X 0,Y 55.269,Z 527.702,A -85,B 0,C 180,E1 -29039.435,E2 -29039.435} C_VEL
LIN {X 0,Y 52.495,Z 529.108,A -85,B 0,C 180,E1 -29046.328,E2 -29046.328} C_VEL
LIN {X 0,Y 49.279,Z 530.695,A -85,B 0,C 180,E1 -29061.809,E2 -29061.809} C_VEL
LIN {X 0,Y 48.886,Z 530.92,A -85,B 0,C 180,E1 -29070.008,E2 -29070.008} C_VEL
LIN {X 0,Y 49.278,Z 530.72,A -85,B 0,C 180,E1 -29078.208,E2 -29078.208} C_VEL
LIN {X 0,Y 52.453,Z 529.169,A -85,B 0,C 180,E1 -29093.709,E2 -29093.709} C_VEL
LIN {X 0,Y 55.21,Z 527.797,A -85,B 0,C 180,E1 -29100.618,E2 -29100.618} C_VEL
LIN {X 0,Y 60.578,Z 524.916,A -85,B 0,C 180,E1 -29109.658,E2 -29109.658} C_VEL
LIN {X 0,Y 67.137,Z 520.991,A -85,B 0,C 180,E1 -29117.128,E2 -29117.128} C_VEL
LIN {X 0,Y 74.573,Z 515.901,A -85,B 0,C 180,E1 -29123.241,E2 -29123.241} C_VEL
LIN {X 0,Y 82.718,Z 509.476,A -85,B 0,C 180,E1 -29128.18,E2 -29128.18} C_VEL
LIN {X 0,Y 85.571,Z 507.016,A -85,B 0,C 180,E1 -29129.592,E2 -29129.592} C_VEL
LIN {X 0,Y 86.942,Z 505.371,A -85,B 0,C 180,E1 -29130.986,E2 -29130.986} C_VEL
LIN {X 0,Y 73.335,Z 510.474,A -85,B 0,C 180,E1 -29143.423,E2 -29143.423} C_VEL
LIN {X 0,Y 63.278,Z 518.851,A -85,B 0,C 180,E1 -29179.463,E2 -29179.463} C_VEL
LIN {X 0,Y 70.237,Z 522.32,A -85,B 0,C 180,E1 -29198.585,E2 -29198.585} C_VEL
LIN {X 0,Y 69.189,Z 523.682,A -85,B 0,C 180,E1 -29201.054,E2 -29201.054} C_VEL
LIN {X 0,Y 62.2,Z 527.796,A -85,B 0,C 180,E1 -29207.308,E2 -29207.308} C_VEL
LIN {X 0,Y 58.034,Z 530.106,A -85,B 0,C 180,E1 -29212.726,E2 -29212.726} C_VEL
LIN {X 0,Y 54.482,Z 531.991,A -85,B 0,C 180,E1 -29218.928,E2 -29218.928} C_VEL
LIN {X 0,Y 51.69,Z 533.414,A -85,B 0,C 180,E1 -29225.919,E2 -29225.919} C_VEL
LIN {X 0,Y 48.802,Z 535.053,A -85,B 0,C 180,E1 -29241.712,E2 -29241.712} C_VEL
LIN {X 0,Y 48.649,Z 535.277,A -85,B 0,C 180,E1 -29249.992,E2 -29249.992} C_VEL
LIN {X 0,Y 48.568,Z 535.023,A -85,B 0,C 180,E1 -29258.312,E2 -29258.312} C_VEL
LIN {X 0,Y 51.002,Z 533.333,A -85,B 0,C 180,E1 -29274.409,E2 -29274.409} C_VEL
LIN {X 0,Y 53.519,Z 531.867,A -85,B 0,C 180,E1 -29281.678,E2 -29281.678} C_VEL
LIN {X 0,Y 58.819,Z 528.859,A -85,B 0,C 180,E1 -29291.075,E2 -29291.075} C_VEL
LIN {X 0,Y 67.103,Z 523.631,A -85,B 0,C 180,E1 -29300.416,E2 -29300.416} C_VEL
LIN {X 0,Y 75.527,Z 517.53,A -85,B 0,C 180,E1 -29306.864,E2 -29306.864} C_VEL
LIN {X 0,Y 83.919,Z 510.439,A -85,B 0,C 180,E1 -29311.553,E2 -29311.553} C_VEL
LIN {X 0,Y 92.828,Z 501.626,A -85,B 0,C 180,E1 -29315.29,E2 -29315.29} C_VEL
LIN {X 0,Y 100.573,Z 492.586,A -85,B 0,C 180,E1 -29317.794,E2 -29317.794} C_VEL
LIN {X 0,Y 107.653,Z 482.531,A -85,B 0,C 180,E1 -29319.782,E2 -29319.782} C_VEL
LIN {X 0,Y 114.068,Z 471.406,A -85,B 0,C 180,E1 -29321.302,E2 -29321.302} C_VEL
LIN {X 0,Y 119.296,Z 460.021,A -85,B 0,C 180,E1 -29322.393,E2 -29322.393} C_VEL
LIN {X 0,Y 123.619,Z 447.488,A -85,B 0,C 180,E1 -29323.209,E2 -29323.209} C_VEL
LIN {X 0,Y 126.705,Z 434.274,A -85,B 0,C 180,E1 -29323.82,E2 -29323.82} C_VEL
LIN {X 0,Y 128.191,Z 423.544,A -85,B 0,C 180,E1 -29324.192,E2 -29324.192} C_VEL
LIN {X 0,Y 126.684,Z 419.406,A -85,B 0,C 180,E1 -29327.79,E2 -29327.79} C_VEL
LIN {X 0,Y 125.345,Z 415.722,A -85,B 0,C 180,E1 -29332.348,E2 -29332.348} C_VEL
LIN {X 0,Y 124.625,Z 412.465,A -85,B 0,C 180,E1 -29338.384,E2 -29338.384} C_VEL
LIN {X 0,Y 124.622,Z 412.708,A -85,B 0,C 180,E1 -29342.424,E2 -29342.424} C_VEL
LIN {X 0,Y 125.671,Z 416.659,A -85,B 0,C 180,E1 -29349.455,E2 -29349.455} C_VEL
LIN {X 0,Y 126.988,Z 420.309,A -85,B 0,C 180,E1 -29353.502,E2 -29353.502} C_VEL
LIN {X 0,Y 128.252,Z 423.957,A -85,B 0,C 180,E1 -29356.484,E2 -29356.484} C_VEL
LIN {X 0,Y 126.021,Z 436.887,A -85,B 0,C 180,E1 -29357.048,E2 -29357.048} C_VEL
LIN {X 0,Y 123.785,Z 444.427,A -85,B 0,C 180,E1 -29356.991,E2 -29356.991} C_VEL
LIN {X 0,Y 120.825,Z 451.703,A -85,B 0,C 180,E1 -29356.428,E2 -29356.428} C_VEL
LIN {X 0,Y 116.591,Z 460.606,A -85,B 0,C 180,E1 -29355.919,E2 -29355.919} C_VEL
LIN {X 0,Y 113.993,Z 465.847,A -85,B 0,C 180,E1 -29356.166,E2 -29356.166} C_VEL
LIN {X 0,Y 107.806,Z 476.952,A -85,B 0,C 180,E1 -29357.569,E2 -29357.569} C_VEL
LIN {X 0,Y 100.617,Z 487.355,A -85,B 0,C 180,E1 -29359.458,E2 -29359.458} C_VEL
LIN {X 0,Y 92.809,Z 496.726,A -85,B 0,C 180,E1 -29361.943,E2 -29361.943} C_VEL
LIN {X 0,Y 83.706,Z 505.723,A -85,B 0,C 180,E1 -29365.514,E2 -29365.514} C_VEL
LIN {X 0,Y 74.866,Z 512.947,A -85,B 0,C 180,E1 -29369.745,E2 -29369.745} C_VEL
LIN {X 0,Y 65.146,Z 519.564,A -85,B 0,C 180,E1 -29376.003,E2 -29376.003} C_VEL
LIN {X 0,Y 57.641,Z 523.894,A -85,B 0,C 180,E1 -29382.993,E2 -29382.993} C_VEL
LIN {X 0,Y 53.2,Z 526.167,A -85,B 0,C 180,E1 -29388.67,E2 -29388.67} C_VEL
LIN {X 0,Y 49.282,Z 528.02,A -85,B 0,C 180,E1 -29395.23,E2 -29395.23} C_VEL
LIN {X 0,Y 46.095,Z 529.424,A -85,B 0,C 180,E1 -29402.79,E2 -29402.79} C_VEL
LIN {X 0,Y 42.282,Z 531.012,A -85,B 0,C 180,E1 -29420.442,E2 -29420.442} C_VEL
LIN {X 0,Y 41.805,Z 531.237,A -85,B 0,C 180,E1 -29430.01,E2 -29430.01} C_VEL
LIN {X 0,Y 42.281,Z 531.036,A -85,B 0,C 180,E1 -29439.578,E2 -29439.578} C_VEL
LIN {X 0,Y 46.042,Z 529.485,A -85,B 0,C 180,E1 -29457.263,E2 -29457.263} C_VEL
LIN {X 0,Y 49.235,Z 528.114,A -85,B 0,C 180,E1 -29464.828,E2 -29464.828} C_VEL
LIN {X 0,Y 55.304,Z 525.231,A -85,B 0,C 180,E1 -29474.352,E2 -29474.352} C_VEL
LIN {X 0,Y 62.515,Z 521.306,A -85,B 0,C 180,E1 -29481.911,E2 -29481.911} C_VEL
LIN {X 0,Y 70.558,Z 516.214,A -85,B 0,C 180,E1 -29487.859,E2 -29487.859} C_VEL
LIN {X 0,Y 76.013,Z 512.28,A -85,B 0,C 180,E1 -29490.968,E2 -29490.968} C_VEL
LIN {X 0,Y 76.428,Z 511.474,A -85,B 0,C 180,E1 -29492.627,E2 -29492.627} C_VEL
LIN {X 0,Y 60.768,Z 517.213,A -85,B 0,C 180,E1 -29513.358,E2 -29513.358} C_VEL
LIN {X 0,Y 57.177,Z 522.161,A -85,B 0,C 180,E1 -29541.638,E2 -29541.638} C_VEL
LIN {X 0,Y 62.367,Z 524.715,A -85,B 0,C 180,E1 -29557.916,E2 -29557.916} C_VEL
LIN {X 0,Y 54.814,Z 528.716,A -85,B 0,C 180,E1 -29565.145,E2 -29565.145} C_VEL
LIN {X 0,Y 48.529,Z 531.674,A -85,B 0,C 180,E1 -29574.59,E2 -29574.59} C_VEL
LIN {X 0,Y 45.308,Z 533.098,A -85,B 0,C 180,E1 -29582.257,E2 -29582.257} C_VEL
LIN {X 0,Y 41.775,Z 534.736,A -85,B 0,C 180,E1 -29600.305,E2 -29600.305} C_VEL
LIN {X 0,Y 41.54,Z 534.96,A -85,B 0,C 180,E1 -29609.99,E2 -29609.99} C_VEL
LIN {X 0,Y 41.531,Z 534.705,A -85,B 0,C 180,E1 -29619.733,E2 -29619.733} C_VEL
LIN {X 0,Y 44.605,Z 533.014,A -85,B 0,C 180,E1 -29638.198,E2 -29638.198} C_VEL
LIN {X 0,Y 47.587,Z 531.547,A -85,B 0,C 180,E1 -29646.2,E2 -29646.2} C_VEL
LIN {X 0,Y 53.646,Z 528.54,A -85,B 0,C 180,E1 -29656.088,E2 -29656.088} C_VEL
LIN {X 0,Y 60.924,Z 524.475,A -85,B 0,C 180,E1 -29663.84,E2 -29663.84} C_VEL
LIN {X 0,Y 70.447,Z 518.221,A -85,B 0,C 180,E1 -29670.787,E2 -29670.787} C_VEL
LIN {X 0,Y 79.258,Z 511.417,A -85,B 0,C 180,E1 -29675.34,E2 -29675.34} C_VEL
LIN {X 0,Y 86.95,Z 504.482,A -85,B 0,C 180,E1 -29678.346,E2 -29678.346} C_VEL
LIN {X 0,Y 94.866,Z 496.121,A -85,B 0,C 180,E1 -29680.819,E2 -29680.819} C_VEL
LIN {X 0,Y 102.961,Z 485.788,A -85,B 0,C 180,E1 -29682.853,E2 -29682.853} C_VEL
LIN {X 0,Y 110.342,Z 474.175,A -85,B 0,C 180,E1 -29684.427,E2 -29684.427} C_VEL
LIN {X 0,Y 116.142,Z 462.512,A -85,B 0,C 180,E1 -29685.495,E2 -29685.495} C_VEL
LIN {X 0,Y 120.819,Z 450.204,A -85,B 0,C 180,E1 -29686.272,E2 -29686.272} C_VEL
LIN {X 0,Y 124.199,Z 437.722,A -85,B 0,C 180,E1 -29686.803,E2 -29686.803} C_VEL
LIN {X 0,Y 125.889,Z 427.71,A -85,B 0,C 180,E1 -29687.199,E2 -29687.199} C_VEL
LIN {X 0,Y 124.821,Z 424.379,A -85,B 0,C 180,E1 -29690.684,E2 -29690.684} C_VEL
LIN {X 0,Y 124.286,Z 422.539,A -85,B 0,C 180,E1 -29693.099,E2 -29693.099} C_VEL
LIN {X 0,Y 123.721,Z 419.473,A -85,B 0,C 180,E1 -29699.186,E2 -29699.186} C_VEL
LIN {X 0,Y 123.726,Z 419.658,A -85,B 0,C 180,E1 -29701.831,E2 -29701.831} C_VEL
LIN {X 0,Y 124.51,Z 423.372,A -85,B 0,C 180,E1 -29708.521,E2 -29708.521} C_VEL
LIN {X 0,Y 125.464,Z 426.641,A -85,B 0,C 180,E1 -29712.229,E2 -29712.229} C_VEL
LIN {X 0,Y 125.855,Z 428.019,A -85,B 0,C 180,E1 -29713.497,E2 -29713.497} C_VEL
LIN {X 0,Y 123.186,Z 441.088,A -85,B 0,C 180,E1 -29714.112,E2 -29714.112} C_VEL
LIN {X 0,Y 119.179,Z 453.724,A -85,B 0,C 180,E1 -29714.969,E2 -29714.969} C_VEL
LIN {X 0,Y 113.993,Z 465.847,A -85,B 0,C 180,E1 -29716.166,E2 -29716.166} C_VEL
LIN {X 0,Y 111.161,Z 471.003,A -85,B 0,C 180,E1 -29716.447,E2 -29716.447} C_VEL
LIN {X 0,Y 105.542,Z 479.148,A -85,B 0,C 180,E1 -29716.092,E2 -29716.092} C_VEL
LIN {X 0,Y 99.316,Z 486.84,A -85,B 0,C 180,E1 -29715.805,E2 -29715.805} C_VEL
LIN {X 0,Y 95.525,Z 491.286,A -85,B 0,C 180,E1 -29716.298,E2 -29716.298} C_VEL
LIN {X 0,Y 87.028,Z 500.451,A -85,B 0,C 180,E1 -29718.846,E2 -29718.846} C_VEL
LIN {X 0,Y 77.8,Z 508.637,A -85,B 0,C 180,E1 -29722.207,E2 -29722.207} C_VEL
LIN {X 0,Y 70.085,Z 514.343,A -85,B 0,C 180,E1 -29725.526,E2 -29725.526} C_VEL
LIN {X 0,Y 61.239,Z 519.881,A -85,B 0,C 180,E1 -29730.615,E2 -29730.615} C_VEL
LIN {X 0,Y 53.058,Z 524.211,A -85,B 0,C 180,E1 -29737.381,E2 -29737.381} C_VEL
LIN {X 0,Y 48.089,Z 526.485,A -85,B 0,C 180,E1 -29743.065,E2 -29743.065} C_VEL
LIN {X 0,Y 43.64,Z 528.337,A -85,B 0,C 180,E1 -29749.909,E2 -29749.909} C_VEL
LIN {X 0,Y 39.915,Z 529.742,A -85,B 0,C 180,E1 -29758.127,E2 -29758.127} C_VEL
LIN {X 0,Y 35.306,Z 531.329,A -85,B 0,C 180,E1 -29778.53,E2 -29778.53} C_VEL
LIN {X 0,Y 34.727,Z 531.553,A -85,B 0,C 180,E1 -29790.012,E2 -29790.012} C_VEL
LIN {X 0,Y 35.305,Z 531.353,A -85,B 0,C 180,E1 -29801.494,E2 -29801.494} C_VEL
LIN {X 0,Y 39.858,Z 529.802,A -85,B 0,C 180,E1 -29821.948,E2 -29821.948} C_VEL
